objectList.M_GetIterator(iter);
WHILE iter.pNode > 0 AND_THEN iter.pNode^.P_pObject > 0 DO
	pObject := iter.pNode^.P_pObject;
	id := pObject^.P_nObjectID;
	a_pObjects[id] := 0;
	pObject^.M_ClearAllProps(TRUE);
	CASE pObject^.P_eObjectType OF
		E_ObjectType.OBJECTTYPE_Cartridge:
			pCartridge := pObject;
			__DELETE(pCartridge);
		E_ObjectType.OBJECTTYPE_FlipTube:
			pFlipTube := pObject;
			__DELETE(pFlipTube);
		E_ObjectType.OBJECTTYPE_Mtp:
			pMtp := pObject;
			__DELETE(pMtp);
		E_ObjectType.OBJECTTYPE_Needle:
			pNeedle := pObject;
			__DELETE(pNeedle);
		E_ObjectType.OBJECTTYPE_Nozzle:
			pNozzle := pObject;
			__DELETE(pNozzle);		
		E_ObjectType.OBJECTTYPE_pHElectrodeCap:
			pPHElectrodeCap := pObject;
			__DELETE(pPHElectrodeCap);
		E_ObjectType.OBJECTTYPE_Point:
			pPoint := pObject;
			__DELETE(pPoint);
		E_ObjectType.OBJECTTYPE_Port:
			pPort := pObject;
			__DELETE(pPort);
		E_ObjectType.OBJECTTYPE_Septum:
			pSeptum := pObject;
			__DELETE(pSeptum);
		E_ObjectType.OBJECTTYPE_Slide:
			pSlide := pObject;
			__DELETE(pSlide);
		E_ObjectType.OBJECTTYPE_SpotArray:
			pSpotArray := pObject;
			__DELETE(pSpotArray);
		(*E_ObjectType.OBJECTTYPE_SpotPattern:
			pSpotPattern := pObject;
			__DELETE(pSpotPattern);*)
		E_ObjectType.OBJECTTYPE_Stamp:
			pStamp := pObject;
			__DELETE(pStamp);
		E_ObjectType.OBJECTTYPE_Tip:
			pTip := pObject;
			__DELETE(pTip);
		E_ObjectType.OBJECTTYPE_TargetTray:
			pTray := pObject;
			__DELETE(pTray);
		E_ObjectType.OBJECTTYPE_Vial:
			pVial := pObject;
			__DELETE(pVial);
		E_ObjectType.OBJECTTYPE_VialClosed:
			pVialClosed := pObject;
			__DELETE(pVialClosed);
		(*E_ObjectType.OBJECTTYPE_Wafer:
			pWafer := pObject;
			__DELETE(pWafer);	*)
	END_CASE
	iter.M_Increment();
END_WHILE

objectList.M_Clear();
fbIdPool.M_Reset();
deviceList.M_Clear();

fbConfiguration.M_Deactivate();

FOR i := 1 TO cMaxMzHeads BY 1 DO
	aFbMultiZRef[i].M_DelConfig();
END_FOR
END_METHOD

METHOD M_DeleteObject : E_ErrorIdObjMgmt
VAR_INPUT
	nObjectID		: UINT;
END_VAR
VAR
	pDeviceNode	: POINTER TO FB_ObjCollectionNode;
	iter : FB_ObjCollectIterator;
END_VAR
//Existiert das Objekt ?
IF nObjectID > 0 AND nObjectID <= cMaxObjects THEN
	IF a_pObjects[nObjectId] > 0 THEN
		//Es können nur Objekte ohne Childs gelöscht werden
		IF NOT a_pObjects[nObjectId]^.P_bHasChilds THEN
			IF a_pObjects[nObjectId]^.M_bIsGroup(E_ObjectGroup.OBJECTGROUP_Device) THEN
				deviceList.M_GetIterator(iter);
				WHILE iter.pNode > 0 DO
					IF iter.pNode^.P_pObject = a_pObjects[nObjectId] THEN
						deviceList.M_ClearNode(iter.pNode);
						EXIT;
					END_IF
					iter.M_Increment();
				END_WHILE
			END_IF
		
			IF a_pObjects[nObjectId]^.P_nNotifyId > 0 THEN
				nCntNotifiIds := nCntNotifiIds - 1;
			END_IF
		
			IF a_pObjects[nObjectId]^.P_pParentObject > 0 THEN
				a_pObjects[nObjectId]^.P_pParentObject^.M_RemoveChild(a_pObjects[nObjectId]);
			ELSE
				IF a_pObjects[nObjectId]^.P_pObjCollectNode > 0 THEN
					a_pObjects[nObjectId]^.P_pObjCollectNode^.P_pOwnerColl^.M_ClearNode(a_pObjects[nObjectId]^.P_pObjCollectNode);
				END_IF
			END_IF
			
			IF a_pObjects[nObjectId]^.M_bIsGroup(E_ObjectGroup.OBJECTGROUP_MzTool) THEN
				fbConfiguration.M_Deactivate();
			END_IF
 			
			a_pObjects[nObjectId]^.M_ClearAllProps(FALSE);
		
			nCntObject := nCntObject - 1;
			
			CASE a_pObjects[nObjectId]^.P_eObjectType OF
				E_ObjectType.OBJECTTYPE_MZHead:
					nCntMZHead := nCntMZHead - 1;
				E_ObjectType.OBJECTTYPE_PiezoPip:
					nCntPiezoPip := nCntPiezoPip - 1;
				E_ObjectType.OBJECTTYPE_PassivPip:
					nCntPassivPip := nCntPassivPip - 1;
				E_ObjectType.OBJECTTYPE_pHElectrode:
					nCntpHElectrode := nCntpHElectrode - 1;
				E_ObjectType.OBJECTTYPE_pHElectrodeCap:
					pPHElectrodeCap := a_pObjects[nObjectId];
					__DELETE(pPHElectrodeCap);
				E_ObjectType.OBJECTTYPE_pHElectrodeCapRack:
					nCntpHElectrodeCapRack := nCntpHElectrodeCapRack - 1;
				E_ObjectType.OBJECTTYPE_PowderPip:
					nCntPowderPip := nCntPowderPip - 1;
				E_ObjectType.OBJECTTYPE_MultiCartHolder:
					nCntMultiCartHolder := nCntMultiCartHolder - 1;
				E_ObjectType.OBJECTTYPE_HybridDispenser:
					nCntHybridDispenser := nCntHybridDispenser - 1;
				E_ObjectType.OBJECTTYPE_CartDispenser:
					nCntCartDispenser := nCntCartDispenser - 1;
				E_ObjectType.OBJECTTYPE_CartDispStirrer:
					nCntCartDispStirrer := nCntCartDispStirrer - 1;
				E_ObjectType.OBJECTTYPE_CartHolder:
					nCntCartHolder := nCntCartHolder - 1;
				E_ObjectType.OBJECTTYPE_Camera:
					nCntCamera := nCntCamera - 1;
				E_ObjectType.OBJECTTYPE_ZSensor:
					nCntZLevelSensor := nCntZLevelSensor - 1;
				E_ObjectType.OBJECTTYPE_StampSupport:
					nCntStampSupport := nCntStampSupport - 1;
				E_ObjectType.OBJECTTYPE_Luer:
					nCntLuer := nCntLuer - 1;
				E_ObjectType.OBJECTTYPE_TrayTransporter:
					nCntTrayTransporter := nCntTrayTransporter - 1;
				E_ObjectType.OBJECTTYPE_TriplePip:
					nCntTriplePip := nCntTriplePip - 1;
				E_ObjectType.OBJECTTYPE_VacuumHandler:
					nCntVacuumHandler := nCntVacuumHandler - 1;
				E_ObjectType.OBJECTTYPE_Workplate:
					nCntWorkplate := nCntWorkplate - 1;
				E_ObjectType.OBJECTTYPE_TipCleaner:
					nCntTipCleaner := nCntTipCleaner - 1;
				E_ObjectType.OBJECTTYPE_TipCleanerGen2:
					nCntTipCleanerGen2 := nCntTipCleanerGen2 - 1;
				E_ObjectType.OBJECTTYPE_TipCalibrator:
					nCntTipCalibrator := nCntTipCalibrator - 1;
				E_ObjectType.OBJECTTYPE_TitrationTool:
					nCntTitrationTool := nCntTitrationTool - 1;
				E_ObjectType.OBJECTTYPE_WashStation:
					nCntWashStation := nCntWashStation - 1;
				E_ObjectType.OBJECTTYPE_LiquidReserve:
					nCntLiquidReserve := nCntLiquidReserve - 1;
				E_ObjectType.OBJECTTYPE_DryPad:
					nCntDrayPad := nCntDrayPad - 1;
				E_ObjectType.OBJECTTYPE_Stroboscope:
					nCntStroboscope := nCntStroboscope - 1;
				E_ObjectType.OBJECTTYPE_MtpHolder:
					nCntMtpHolder := nCntMtpHolder - 1;
				E_ObjectType.OBJECTTYPE_SubstHolder:
					nCntSubstHolder := nCntSubstHolder - 1;
				E_ObjectType.OBJECTTYPE_SubstHolderUnistat:
					nCntSubstHolderUnistat := nCntSubstHolderUnistat - 1;
				E_ObjectType.OBJECTTYPE_StampMagazine:
					nCntStampMagazine := nCntStampMagazine - 1;
				E_ObjectType.OBJECTTYPE_InkStation:
					nCntInkStation := nCntInkStation - 1;
				E_ObjectType.OBJECTTYPE_PowderStation:
					nCntPowderStation := nCntPowderStation - 1;
				E_ObjectType.OBJECTTYPE_Reactor:
					nCntReactor := nCntReactor - 1;
				E_ObjectType.OBJECTTYPE_TargetTray:
					pTray := a_pObjects[nObjectId];
					__DELETE(pTray);
				E_ObjectType.OBJECTTYPE_SpotArray:
					pSpotArray := a_pObjects[nObjectId];
					__DELETE(pSpotArray);
				E_ObjectType.OBJECTTYPE_Mtp:
					pMtp := a_pObjects[nObjectId];
					__DELETE(pMtp);
				E_ObjectType.OBJECTTYPE_Slide:
					pSlide := a_pObjects[nObjectId];
					__DELETE(pSlide);
				(*E_ObjectType.OBJECTTYPE_Wafer:
					pWafer := a_pObjects[nObjectId];
					__DELETE(pWafer);	*)				
				E_ObjectType.OBJECTTYPE_Point:
					pPoint := a_pObjects[nObjectId];
					__DELETE(pPoint);
				E_ObjectType.OBJECTTYPE_Diluter:
					fbConfiguration.M_Deactivate();
					nCntDiluter := nCntDiluter - 1;
				E_ObjectType.OBJECTTYPE_Diluter3Inputs:
					fbConfiguration.M_Deactivate();
					nCntDiluter3Inputs := nCntDiluter3Inputs - 1;
				(*E_ObjectType.OBJECTTYPE_SpotPattern:
					pSpotPattern := a_pObjects[nObjectId];
					__DELETE(pSpotPattern);*)
				E_ObjectType.OBJECTTYPE_DeloDot:
					nCntDeloDot := nCntDeloDot - 1;
				E_ObjectType.OBJECTTYPE_Exposure:
					nCntExposure := nCntExposure - 1;
				E_ObjectType.OBJECTTYPE_Stamp:
					pStamp := a_pObjects[nObjectId];
					__DELETE(pStamp);
				E_ObjectType.OBJECTTYPE_Needle:
					pNeedle := a_pObjects[nObjectId];
					__DELETE(pNeedle);
				E_ObjectType.OBJECTTYPE_Tip:
					pTip := a_pObjects[nObjectId];
					__DELETE(pTip);
				E_ObjectType.OBJECTTYPE_Vial:
					pVial := a_pObjects[nObjectId];
					__DELETE(pVial);
				E_ObjectType.OBJECTTYPE_VialClosed:
					pVialClosed := a_pObjects[nObjectId];
					__DELETE(pVialClosed);
				E_ObjectType.OBJECTTYPE_Septum:
					pSeptum := a_pObjects[nObjectId];
					__DELETE(pSeptum);
				E_ObjectType.OBJECTTYPE_Cartridge:
					pCartridge := a_pObjects[nObjectId];
					__DELETE(pCartridge);
				E_ObjectType.OBJECTTYPE_Port:
					pPort := a_pObjects[nObjectId];
					__DELETE(pPort);
				E_ObjectType.OBJECTTYPE_FlipTube:
					pFlipTube := a_pObjects[nObjectId];
					__DELETE(pFlipTube);
				E_ObjectType.OBJECTTYPE_SeptumWaste:
					nCntSeptumWaste := nCntSeptumWaste - 1;
				E_ObjectType.OBJECTTYPE_NeedleRack:
					nCntNeedleRack := nCntNeedleRack - 1;
				E_ObjectType.OBJECTTYPE_TipRack:
					nCntTipRack := nCntTipRack - 1;
				E_ObjectType.OBJECTTYPE_FlipTubeRack:
					nCntFlipTubeRack := nCntFlipTubeRack - 1;
				E_ObjectType.OBJECTTYPE_SeptumRack:
					nCntSeptumRack := nCntSeptumRack - 1;
				E_ObjectType.OBJECTTYPE_VialRack:
					nCntVialRack := nCntVialRack - 1;
				E_ObjectType.OBJECTTYPE_PortRack:
					nCntPortRack := nCntPortRack - 1;
				E_ObjectType.OBJECTTYPE_Nozzle:
					fbConfiguration.M_Deactivate();
					pNozzle := a_pObjects[nObjectId];
					__DELETE(pNozzle);
				E_ObjectType.OBJECTTYPE_SinglePiezoHolder:
					nCntSinglePiezoHolder := nCntSinglePiezoHolder - 1;
				E_ObjectType.OBJECTTYPE_TwinPiezoHolder:
					nCntTwinPiezoHolder := nCntTwinPiezoHolder - 1;
				E_ObjectType.OBJECTTYPE_HighVoltTray:
					nCntHighVoltTray := nCntHighVoltTray - 1;
				E_ObjectType.OBJECTTYPE_SolenoidPip:
					nCntSolenoidPip := nCntSolenoidPip - 1;
				E_ObjectType.OBJECTTYPE_Extruder:
					nCntExtruder := nCntExtruder - 1;
				E_ObjectType.OBJECTTYPE_TwinExtruder:
					nCntTwinExtruder := nCntTwinExtruder - 1;
				E_ObjectType.OBJECTTYPE_VermesDisp:
					nCntVermesDisp := nCntVermesDisp - 1;
				E_ObjectType.OBJECTTYPE_WorkplateCamera:
					nCntWorkplateCamera := nCntWorkplateCamera - 1;
				E_ObjectType.OBJECTTYPE_DummyTool:
					nCntDummyTool := nCntDummyTool - 1;
				E_ObjectType.OBJECTTYPE_CustomUnitType1:
					nCntCustomUnitType1 := nCntCustomUnitType1 - 1;
				E_ObjectType.OBJECTTYPE_CustomUnitType2:
					nCntCustomUnitType2 := nCntCustomUnitType2 - 1;
				E_ObjectType.OBJECTTYPE_Gripper:
					nCntGripper := nCntGripper - 1;
				E_ObjectType.OBJECTTYPE_PickPlacePip:
					nCntPickPlacePip := nCntPickPlacePip - 1;
				E_ObjectType.OBJECTTYPE_Stacker:
					nCntStacker := nCntStacker - 1;
			END_CASE
			a_pObjects[nObjectId] := 0;
			//ObjectID wieder freigeben
			fbIdPool.M_ReleaseId(nObjectId);
		ELSE
			M_DeleteObject := E_ErrorIdObjMgmt.ERRORID_ObjectHasChilds;
		END_IF
	ELSE
		M_DeleteObject := E_ErrorIdObjMgmt.ERRORID_InvalidObjectId;
	END_IF
END_IF
END_METHOD

METHOD M_GetChangedObjId : UINT
VAR_INPUT
END_VAR
IF hList.nCount > 0 THEN
	fbList.A_GetTail(hList:= hList);
	{IF hasvalue (RegisterSize, '32')}
	M_GetChangedObjId := UDINT_TO_UINT(fbList.getValue);
	{ELSE}
	M_GetChangedObjId := ULINT_TO_UINT(fbList.getValue);
	{END_IF}
	fbList.A_RemoveTailValue(hList:= hList);
END_IF
END_METHOD

METHOD M_GetCoHead : POINTER TO FB_MzHead
VAR_INPUT
	pMzHead : POINTER TO FB_MzHead;
END_VAR

VAR
	i : UINT;
END_VAR
FOR i:= 1 TO nCntMZHead BY 1 DO
	IF ADR(afbMzHead[i]) <> pMzHead THEN
		IF afbMzHead[i].P_eObjectType = E_ObjectType.OBJECTTYPE_MZHead THEN
			IF afbMzHead[i].P_pXDrive = pMzHead^.P_pXDrive THEN
				M_GetCoHead := ADR(afbMzHead[i]);
			END_IF
		END_IF
	END_IF
END_FOR
END_METHOD

METHOD M_GetConfigCheckSum : UINT
VAR_INPUT
END_VAR

VAR
	nObjectCounter 	: UINT;
	wPrevious 		: WORD := 16#FFFF;
	iter			: FB_ObjCollectIteratorDeep;
	nLevel			: UINT;
	nObjType		: UINT;
	nNoOfProps		: UINT;
	nParentSlotNr	: UINT;
END_VAR
objectList.M_GetIterator(iter);
WHILE iter.pNode > 0 AND_THEN iter.pNode^.P_pObject > 0 DO
	
	nParentSlotNr := iter.pNode^.P_pObject^.P_nParentSlotNr;
	wPrevious := F_DATA_TO_CRC16_CCITT(ADR(nParentSlotNr),SIZEOF(nParentSlotNr),wPrevious);

	nLevel := iter.pNode^.M_GetLevel(0);
	wPrevious := F_DATA_TO_CRC16_CCITT(ADR(nLevel),SIZEOF(nLevel),wPrevious); 

	nObjType := iter.pNode^.P_pObject^.P_eObjectType;
	wPrevious := F_DATA_TO_CRC16_CCITT(ADR(nObjType),SIZEOF(nObjType),wPrevious);

	nNoOfProps := iter.pNode^.P_pObject^.P_nNoOfProps;
	wPrevious := F_DATA_TO_CRC16_CCITT(ADR(nNoOfProps),SIZEOF(nNoOfProps),wPrevious);

	iter.M_Increment();
END_WHILE
M_GetConfigCheckSum := WORD_TO_UINT(wPrevious);
END_METHOD

METHOD M_GetDevice : I_Device
VAR_INPUT
	nObjectId : UINT;
END_VAR

VAR
	pActiveTarget : POINTER TO FB_ActiveTarget;
	pMzToolBase	: POINTER TO FB_MzBase;
	pDiluter : POINTER TO FB_Diluter; 
END_VAR
IF M_ObjIsDevice(nObjectId) THEN
	M_GetDevice := a_pObjects[nObjectId]^.M_GetDevice();
END_IF
END_METHOD

METHOD M_GetObjIdFromGCodeTargetNr : UINT
VAR_INPUT
	nTargetNr : UINT;
END_VAR
END_METHOD

METHOD M_GetObjIdStream : ERRORID
VAR_INPUT
	aData : REFERENCE TO ARRAY[0..999] OF UINT;
END_VAR

VAR
	iter : FB_ObjCollectIteratorDeep;
	i : UINT;
END_VAR
objectList.M_GetIterator(iter);
WHILE iter.pNode > 0 AND_THEN iter.pNode^.P_pObject > 0 DO
	IF i > 999 THEN
		M_GetObjIdStream := 333;
		RETURN;	
	END_IF
	aData[i] := iter.pNode^.P_pObject^.P_nObjectID;
	i := i + 1;
	iter.M_Increment();
END_WHILE
END_METHOD

METHOD M_GetObjPointer : POINTER TO FB_Object
VAR_INPUT
	nObjectId : UINT;
END_VAR
IF nObjectId > 0 AND nObjectId <= cMaxObjects THEN
	IF a_pObjects[nObjectId]^.P_nObjectID = nObjectId THEN
		M_GetObjPointer := a_pObjects[nObjectId];
	END_IF
END_IF
END_METHOD

METHOD M_GetObjType : E_ObjectType
VAR_INPUT
	ObjectId	: UINT;
END_VAR
IF ObjectId > 0 AND ObjectId <= cMaxObjects AND_THEN a_pObjects[ObjectId] > 0 THEN
	M_GetObjType := a_pObjects[ObjectId]^.P_eObjectType;
ELSE
	M_GetObjType := E_ObjectType.OBJECTTYPE_UNDEFINED;
END_IF
END_METHOD

METHOD M_GetTipCleaner : POINTER TO FB_TargetBase
VAR_INPUT
END_VAR
//Es wird davon ausgegangen, dass es nur einen TipCleaner in einer Konfiguration gibt.
IF afbTipCleaner[1].P_nObjectID > 0 THEN
	M_GetTipCleaner := ADR(afbTipCleaner[1]);
ELSIF afbTipCleanerGen2[1].P_nObjectID > 0 THEN
	M_GetTipCleaner := ADR(afbTipCleanerGen2[1]);
END_IF
END_METHOD

METHOD M_GetTopHead : POINTER TO FB_MzHead

VAR
	i : UINT;
END_VAR
FOR i:= 1 TO nCntMZHead BY 1 DO
	IF afbMzHead[i].P_bIsTopHead THEN
		M_GetTopHead := ADR(afbMzHead[i]);
		RETURN;
	END_IF
END_FOR
END_METHOD

METHOD M_Init : BOOL
VAR_INPUT
END_VAR

VAR
	i	: UINT;	//allg. Zählveriable
END_VAR
fbIdPool.M_Reset();

F_CreateLinkedListHnd( ADR( nodes ), SIZEOF( nodes ), hList );

bIsInitialized := TRUE;
END_METHOD

METHOD M_MoveObject : ERRORID
VAR_INPUT
	pObject : POINTER TO FB_Object;
	pDestObject : POINTER TO FB_Object;
	nDestSlotNr	: UINT;
END_VAR

VAR
	pSlot : POINTER TO FB_Slot;
END_VAR
//Verschiebt ein Objekt zu einem neuen Objekt oder zu einem anderen Slot.
IF pObject > 0 THEN
	IF pObject^.P_pParentObject > 0 AND_THEN pDestObject > 0 THEN
		IF nDestSlotNr > 0 THEN
			pSlot := pDestObject^.M_GetSlot(nDestSlotNr);
			IF pSlot > 0 THEN
				IF pSlot^.P_pChild > 0 THEN
					M_MoveObject := E_ErrorIdObjMgmt.ERRORID_DestinationSlotNotFree;
					RETURN;
				END_IF
			ELSE
				M_MoveObject := E_ErrorIdObjMgmt.ERRORID_InvalidDestinationSlot;
				RETURN;
			END_IF
		END_IF
		M_MoveObject := pObject^.P_pParentObject^.M_RemoveChild(pObject);
		IF M_MoveObject = 0 THEN
			M_MoveObject := pDestObject^.M_AddChild(pObject,nDestSlotNr,-1);
			//M_SetObjChange(pObject^.P_nObjectID);
			stObjectHasMoved.ObjectId := pObject^.P_nObjectID;
			stObjectHasMoved.DestObjId := pDestObject^.P_nObjectID;
			stObjectHasMoved.DestSlotNr := nDestSlotNr;
			stObjectHasMoved.ChangeCounter := stObjectHasMoved.ChangeCounter + 1;
		END_IF
	ELSE
		M_MoveObject := E_ErrorIdObjMgmt.ERRORID_InvalidObject;
	END_IF
ELSE
	M_MoveObject := E_ErrorIdObjMgmt.ERRORID_InvalidObject;
END_IF
END_METHOD

METHOD M_ObjIsArray : BOOL
VAR_INPUT
	nObjectId	: UINT;
END_VAR
IF nObjectId > 0 AND nObjectId <= cMaxObjects THEN
	IF (a_pObjects[nObjectId]^.P_eObjectGroup AND E_ObjectGroup.OBJECTGROUP_Array) = E_ObjectGroup.OBJECTGROUP_Array THEN
		M_ObjIsArray := TRUE;
	END_IF
END_IF
END_METHOD

METHOD M_ObjIsDevice : BOOL
VAR_INPUT
	nObjectId	: UINT;
END_VAR
IF nObjectId > 0 AND nObjectId <= cMaxObjects THEN
	IF a_pObjects[nObjectId]^.M_bIsGroup(E_ObjectGroup.OBJECTGROUP_Device) THEN
		M_ObjIsDevice := TRUE;
	END_IF
END_IF
END_METHOD

METHOD M_ObjIsGCodeTool : BOOL
VAR_INPUT
	nObjectId	: UINT;
END_VAR
IF nObjectId > 0 AND nObjectId <= cMaxObjects THEN
	IF (a_pObjects[nObjectId]^.P_eObjectGroup AND E_ObjectGroup.OBJECTGROUP_GCodeTool) = E_ObjectGroup.OBJECTGROUP_GCodeTool THEN
		M_ObjIsGCodeTool := TRUE;
	END_IF
END_IF
END_METHOD

METHOD M_ObjIsMzTool : BOOL
VAR_INPUT
	nObjectId	: UINT;
END_VAR
IF nObjectId > 0 AND nObjectId <= cMaxObjects THEN
	IF (a_pObjects[nObjectId]^.P_eObjectGroup AND E_ObjectGroup.OBJECTGROUP_MzTool) = E_ObjectGroup.OBJECTGROUP_MzTool THEN
		M_ObjIsMzTool := TRUE;
	END_IF
END_IF
END_METHOD

METHOD M_ObjIsPiece : BOOL
VAR_INPUT
	nObjectId	: UINT;
END_VAR
IF nObjectId > 0 AND nObjectId <= cMaxObjects THEN
	IF (a_pObjects[nObjectId]^.P_eObjectGroup AND E_ObjectGroup.OBJECTGROUP_Piece) = E_ObjectGroup.OBJECTGROUP_Piece THEN
		M_ObjIsPiece := TRUE;
	END_IF
END_IF
END_METHOD

METHOD M_ObjIsRack : BOOL
VAR_INPUT
	nObjectId	: UINT;
END_VAR
IF nObjectId > 0 AND nObjectId <= cMaxObjects THEN
	IF (a_pObjects[nObjectId]^.P_eObjectGroup AND E_ObjectGroup.OBJECTGROUP_Rack) = E_ObjectGroup.OBJECTGROUP_Rack THEN
		M_ObjIsRack := TRUE;
	END_IF
END_IF
END_METHOD

METHOD M_ObjIsTarget : BOOL
VAR_INPUT
	nObjectId	: UINT;
END_VAR
IF nObjectId > 0 AND nObjectId <= cMaxObjects THEN
	IF (a_pObjects[nObjectId]^.P_eObjectGroup AND E_ObjectGroup.OBJECTGROUP_Target) = E_ObjectGroup.OBJECTGROUP_Target THEN
		M_ObjIsTarget := TRUE;
	END_IF
END_IF
END_METHOD

METHOD M_RemoveObjChange
VAR_INPUT
	nObjectId : UINT;
END_VAR

VAR
	getPosPtr : POINTER TO T_LinkedListEntry;
END_VAR
fbList.A_FindNext(hList:= hList, putPosPtr:= 0, putValue:= UINT_TO_UDINT(nObjectId), getPosPtr=> getPosPtr);
IF fbList.bOk THEN //Eintrag vorhanden
	fbList.A_RemoveValueAtPosPtr(hList:= hList, putPosPtr := getPosPtr);
END_IF
END_METHOD

METHOD M_ResetCustomUnitType2
VAR_INPUT
END_VAR

VAR
	i : UINT;
END_VAR
FOR i := 1 TO nCntCustomUnitType2 DO
	 IF afbCustomUnitType2[i].P_bError THEN
		 afbCustomUnitType2[i].M_Reset();
	 END_IF
END_FOR
END_METHOD

METHOD M_SetObjChange
VAR_INPUT
	nObjectId : UINT;
END_VAR

VAR
	putValue : UDINT;
END_VAR
putValue := UINT_TO_UDINT(nObjectId);
//Checken, ob schon eingetragen
fbList.A_FindNext(hList:= hList, putPosPtr:= 0, putValue:= putValue);
IF NOT fbList.bOk THEN //Eintrag noch nicht vorhanden
	fbList.A_AddHeadValue(hList:= hList, putValue:= putValue);	
	nObjPropChangeCnt := nObjPropChangeCnt + 1;
END_IF
END_METHOD

METHOD M_SetParent : ERRORID
VAR_INPUT
END_VAR
END_METHOD

PROPERTY P_pDeviceCollection : POINTER TO FB_ObjCollection
GET
P_pDeviceCollection := ADR(deviceList);
END_GET
END_PROPERTY

PROPERTY P_pObjectCollection : POINTER TO FB_ObjCollection
GET
P_pObjectCollection := ADR(objectList);
END_GET
END_PROPERTY

END_FUNCTION_BLOCK

// ---- Configuration/FB_IdPool.TcPOU
FUNCTION_BLOCK FB_IdPool
VAR_INPUT
END_VAR
VAR_OUTPUT
END_VAR
VAR
	aNodes : ARRAY[1..cMaxObjects] OF ST_IdNode;
	pHead : POINTER TO ST_IdNode;
	pTail : POINTER TO ST_IdNode;
END_VAR

METHOD M_GetId : UINT
VAR_INPUT
END_VAR

VAR
	pNode : POINTER TO ST_IdNode;
END_VAR
IF pHead > 0 THEN
	pNode := pHead;
	M_GetId := pNode^.nId;
	IF pHead = pTail THEN //die letzte freie Id
		pHead := 0;
		pTail := 0;
	ELSE
		pHead := pNode^.pNext;
	END_IF
	memset(pNode,0,SIZEOF(ST_IdNode));
END_IF
END_METHOD

METHOD M_ReleaseId : BOOL
VAR_INPUT
	nId : UINT;
END_VAR
//Id in Benutzung?
IF nId >= 0 AND nId <= cMaxObjects AND_THEN aNodes[nId].nId = 0 THEN
	aNodes[nId].nId := nId;
	aNodes[nId].pNext := pHead;
	pHead := ADR(aNodes[nId]);
	M_ReleaseId := TRUE;
END_IF
END_METHOD

METHOD M_Reset : BOOL
VAR_INPUT
END_VAR

VAR
	i : UINT;
END_VAR
pHead := ADR(aNodes[1]);
pTail := ADR(aNodes[cMaxObjects]);
FOR i := 1 TO cMaxObjects BY 1 DO
	aNodes[i].nId := i;
	IF i < cMaxObjects THEN
		aNodes[i].pNext := ADR(aNodes[i+1]);
	ELSE
		aNodes[i].pNext := 0;
	END_IF
END_FOR
END_METHOD

END_FUNCTION_BLOCK

// ---- Objects/Pieces/FB_Cartridge.TcPOU
{attribute 'enable_dynamic_creation'}
FUNCTION_BLOCK FB_Cartridge EXTENDS FB_PieceBase
VAR_INPUT
END_VAR
VAR_OUTPUT
END_VAR
VAR
END_VAR

METHOD FB_init : BOOL
VAR_INPUT
	bInitRetains : BOOL; // if TRUE, the retain variables are initialized (warm start / cold start)
	bInCopyCode : BOOL;  // if TRUE, the instance afterwards gets moved into the copy code (online change)
END_VAR
eObjectType := E_ObjectType.OBJECTTYPE_Cartridge;
eObjectGroup := E_ObjectGroup.OBJECTGROUP_Piece;
END_METHOD

END_FUNCTION_BLOCK

// ---- Objects/Pieces/FB_FlipTube.TcPOU
{attribute 'enable_dynamic_creation'}
FUNCTION_BLOCK FB_FlipTube EXTENDS FB_PieceBase
VAR_INPUT
END_VAR
VAR_OUTPUT
END_VAR
VAR
	bIsOpen : BOOL;
	nTopLevel : DINT;
	nBottomLevel : DINT;	
END_VAR

METHOD FB_init : BOOL
VAR_INPUT
	bInitRetains : BOOL; // if TRUE, the retain variables are initialized (warm start / cold start)
	bInCopyCode : BOOL;  // if TRUE, the instance afterwards gets moved into the copy code (online change)
END_VAR
eObjectType := E_ObjectType.OBJECTTYPE_FlipTube;
eObjectGroup := E_ObjectGroup.OBJECTGROUP_Piece;
END_METHOD

METHOD M_GetAllProps : ERRORID
VAR_INPUT
	refCmdData : REFERENCE TO  ST_CmdData;
END_VAR
SUPER^.M_GetAllProps(refCmdData);
nCurrentPropIndex := nCurrentPropIndex + 1;
refCmdData.n32Data[nCurrentPropIndex] := BOOL_TO_DINT(bIsOpen);
nCurrentPropIndex := nCurrentPropIndex + 1;
refCmdData.n32Data[nCurrentPropIndex] := nTopLevel;
nCurrentPropIndex := nCurrentPropIndex + 1;
refCmdData.n32Data[nCurrentPropIndex] := nBottomLevel;
END_METHOD

{attribute 'object_name' := 'M_SetAllProps'}
METHOD M_SetAllProps : ERRORID
VAR_INPUT
	refCmdData	: REFERENCE TO ST_CmdData;
END_VAR
M_SetAllProps := SUPER^.M_SetAllProps(refCmdData);

IF M_SetAllProps > 0 THEN
	RETURN;
END_IF
nCurrentPropIndex := nCurrentPropIndex + 1;
nSpecPropIndex := nCurrentPropIndex;

bIsOpen := DINT_TO_BOOL(refCmdData.n32Data[nCurrentPropIndex]);
nCurrentPropIndex := nCurrentPropIndex + 1;
nTopLevel := refCmdData.n32Data[nCurrentPropIndex];
nCurrentPropIndex := nCurrentPropIndex + 1;
nBottomLevel := refCmdData.n32Data[nCurrentPropIndex];

nNoOfProps := nCurrentPropIndex + 1;
END_METHOD

METHOD M_SetSingleProp : ERRORID
VAR_INPUT
	refCmdData : REFERENCE TO  ST_CmdData;
END_VAR
IF refCmdData.aHeader[1] = nSpecPropIndex THEN
	bIsOpen := DINT_TO_BOOL(refCmdData.n32Data[0]);
ELSIF refCmdData.aHeader[1] + 1 = nSpecPropIndex THEN
	nTopLevel := refCmdData.n32Data[0];
ELSIF refCmdData.aHeader[1] + 2 = nSpecPropIndex THEN
	nBottomLevel := refCmdData.n32Data[0];
ELSE
	M_SetSingleProp := SUPER^.M_SetSingleProp(refCmdData);
END_IF
END_METHOD

PROPERTY P_bIsOpen : BOOL
GET
P_bIsOpen := bIsOpen;
END_GET
SET
bIsOpen := P_bIsOpen;
END_SET
END_PROPERTY

PROPERTY P_nBottomLevel : DINT
GET
P_nBottomLevel := nBottomLevel;
END_GET
END_PROPERTY

PROPERTY P_nTopLevel : DINT
GET
P_nTopLevel := nTopLevel;
END_GET
END_PROPERTY

END_FUNCTION_BLOCK

// ---- Objects/Pieces/FB_Needle.TcPOU
{attribute 'enable_dynamic_creation'}
FUNCTION_BLOCK FB_Needle EXTENDS FB_UsingPiece
VAR_INPUT
END_VAR
VAR_OUTPUT
END_VAR
VAR
	pSeptum : POINTER TO FB_PieceBase;
END_VAR

METHOD FB_init : BOOL
VAR_INPUT
	bInitRetains : BOOL; // if TRUE, the retain variables are initialized (warm start / cold start)
	bInCopyCode : BOOL;  // if TRUE, the instance afterwards gets moved into the copy code (online change)
END_VAR
bUsingPiece := TRUE;
eObjectType := E_ObjectType.OBJECTTYPE_Needle;
eObjectGroup := E_ObjectGroup.OBJECTGROUP_Piece;
END_METHOD

{attribute 'object_name' := 'M_ClearAllProps'}
METHOD M_ClearAllProps

VAR_INPUT
	bIgnoreParent : BOOL; //Es wird das gesamte OD gelöscht. -> Zeiger auf Parent nicht mehr gültig!
END_VAR
pSeptum := 0;
SUPER^.M_ClearAllProps(bIgnoreParent);
END_METHOD

PROPERTY P_pLatestChild : POINTER TO FB_PieceBase
GET
IF pSeptum > 0 THEN
	P_pLatestChild := pSeptum;	
ELSE
	P_pLatestChild := THIS;
END_IF
END_GET
END_PROPERTY

PROPERTY P_pSeptum : POINTER TO FB_PieceBase
GET
P_pSeptum := pSeptum;
END_GET
SET
pSeptum := P_pSeptum;
END_SET
END_PROPERTY

END_FUNCTION_BLOCK

// ---- Objects/Pieces/FB_pHElectrodeCap.TcPOU
{attribute 'enable_dynamic_creation'}
FUNCTION_BLOCK FB_pHElectrodeCap EXTENDS FB_PieceBase
VAR_INPUT
END_VAR
VAR_OUTPUT
END_VAR
VAR
END_VAR

METHOD FB_init : BOOL
VAR_INPUT
	bInitRetains : BOOL; // if TRUE, the retain variables are initialized (warm start / cold start)
	bInCopyCode : BOOL;  // if TRUE, the instance afterwards gets moved into the copy code (online change)
END_VAR
eObjectType := E_ObjectType.OBJECTTYPE_pHElectrodeCap;
eObjectGroup := E_ObjectGroup.OBJECTGROUP_Piece;
END_METHOD

END_FUNCTION_BLOCK

// ---- Objects/Targets/Passive/FB_Point.TcPOU
{attribute 'enable_dynamic_creation'}
FUNCTION_BLOCK FB_Point EXTENDS FB_TargetBase
VAR_INPUT
END_VAR
VAR_OUTPUT
END_VAR
VAR
END_VAR

METHOD FB_init : BOOL
VAR_INPUT
	bInitRetains : BOOL; // if TRUE, the retain variables are initialized (warm start / cold start)
	bInCopyCode : BOOL;  // if TRUE, the instance afterwards gets moved into the copy code (online change)
END_VAR
eObjectType := E_ObjectType.OBJECTTYPE_Point;
eObjectGroup := E_ObjectGroup.OBJECTGROUP_Target;
END_METHOD

METHOD M_AddChild : ERRORID
VAR_INPUT
	pObject : POINTER TO FB_Object;
	nSlotNr	: UINT;
	nIndex 	: INT;
END_VAR
//Kann folgende Objekte aufnehmen:
//Point
IF pObject <> 0 THEN
	IF pObject^.P_eObjectType = E_ObjectType.OBJECTTYPE_Point OR pObject^.P_eObjectType = E_ObjectType.OBJECTTYPE_SpotArray Then
		M_AddChild := SUPER^.M_AddChild(pObject,nSlotNr,nIndex);
	ELSE
		M_AddChild := E_ErrorIdObjMgmt.ERRORID_InvalidParentObject;
	END_IF
ELSE
	M_AddChild := E_ErrorIdObjMgmt.ERRORID_InvalidParentObject;
END_IF
END_METHOD

END_FUNCTION_BLOCK

// ---- Objects/Pieces/FB_Port.TcPOU
{attribute 'enable_dynamic_creation'}
FUNCTION_BLOCK FB_Port EXTENDS FB_PieceBase
VAR_INPUT
END_VAR
VAR_OUTPUT
END_VAR
VAR
END_VAR

METHOD FB_init : BOOL
VAR_INPUT
	bInitRetains : BOOL; // if TRUE, the retain variables are initialized (warm start / cold start)
	bInCopyCode : BOOL;  // if TRUE, the instance afterwards gets moved into the copy code (online change)
END_VAR
eObjectType := E_ObjectType.OBJECTTYPE_Port;
eObjectGroup := E_ObjectGroup.OBJECTGROUP_Piece;
END_METHOD

END_FUNCTION_BLOCK

// ---- Objects/Pieces/FB_Septum.TcPOU
{attribute 'enable_dynamic_creation'}
FUNCTION_BLOCK FB_Septum EXTENDS FB_UsingPiece
VAR_INPUT
END_VAR
VAR_OUTPUT
END_VAR
VAR
	pVial : POINTER TO FB_Vial;
END_VAR

METHOD FB_init : BOOL
VAR_INPUT
	bInitRetains : BOOL; // if TRUE, the retain variables are initialized (warm start / cold start)
	bInCopyCode : BOOL;  // if TRUE, the instance afterwards gets moved into the copy code (online change)
END_VAR
bUsingPiece := TRUE;
eObjectType := E_ObjectType.OBJECTTYPE_Septum;
eObjectGroup := E_ObjectGroup.OBJECTGROUP_Piece;
END_METHOD

{attribute 'object_name' := 'M_ClearAllProps'}
METHOD M_ClearAllProps

VAR_INPUT
	bIgnoreParent : BOOL; //Es wird das gesamte OD gelöscht. -> Zeiger auf Parent nicht mehr gültig!
END_VAR
pVial := 0;
SUPER^.M_ClearAllProps(bIgnoreParent);
END_METHOD

PROPERTY P_pVial : POINTER TO FB_PieceBase
GET
P_pVial := pVial;
END_GET
SET
pVial := P_pVial;
END_SET
END_PROPERTY

END_FUNCTION_BLOCK

// ---- Objects/Targets/Passive/FB_Slide.TcPOU
{attribute 'enable_dynamic_creation'}
FUNCTION_BLOCK FB_Slide EXTENDS FB_TargetBase
VAR_INPUT
END_VAR
VAR_OUTPUT
END_VAR
VAR
	///Spec-Properties TODO: rauslöschen
	(*
	nNoOfSpecPoints: USINT;
	stMark1: ST_3DPoint;
	stMark2: ST_3DPoint;
	stMark1Act: ST_3DPoint;
	stMark2Act: ST_3DPoint;*)
	
	//neue Slide Variablen
	stMarker1Position	: ST_3DPoint;
	stCamOffsetMarker1	: ST_3DPoint;
	stCamOffsetMarker2	: ST_3DPoint;
	rTargetRot			: REAL;			//Winkel * 1000
	
	//ALT: 
	
	lrAngle				: LREAL;
	//bIsAligned			: BOOL;	
END_VAR

METHOD FB_init : BOOL
VAR_INPUT
	bInitRetains : BOOL; // if TRUE, the retain variables are initialized (warm start / cold start)
	bInCopyCode : BOOL;  // if TRUE, the instance afterwards gets moved into the copy code (online change)
END_VAR
eObjectType := E_ObjectType.OBJECTTYPE_Slide;
eObjectGroup := E_ObjectGroup.OBJECTGROUP_Target;
END_METHOD

METHOD M_AddChild : ERRORID
VAR_INPUT
	pObject : POINTER TO FB_Object;
	nSlotNr	: UINT;
	nIndex 	: INT;
END_VAR
//Kann folgende Objekte aufnehmen:
IF pObject > 0 THEN
	IF pObject^.P_eObjectType = E_ObjectType.OBJECTTYPE_Point OR
		pObject^.P_eObjectType = E_ObjectType.OBJECTTYPE_Slide OR
		pObject^.P_eObjectType = E_ObjectType.OBJECTTYPE_Mtp OR
		(*pObject^.P_eObjectType = E_ObjectType.OBJECTTYPE_SpotPattern OR*)
		pObject^.P_eObjectType = E_ObjectType.OBJECTTYPE_SpotArray
		(*pObject^.P_eObjectType = E_ObjectType.OBJECTTYPE_TargetGroup OR
		pObject^.P_eObjectType = E_ObjectType.OBJECTTYPE_Wafer*) THEN
		M_AddChild := SUPER^.M_AddChild(pObject,nSlotNr,nIndex);
	ELSE
		M_AddChild := E_ErrorIdObjMgmt.ERRORID_InvalidParentObject;
	END_IF
ELSE
	M_AddChild := E_ErrorIdObjMgmt.ERRORID_InvalidParentObject;
END_IF
END_METHOD

METHOD M_Align : ST_3DPoint
VAR_INPUT
	stPos: ST_3DPoint;
END_VAR
VAR_OUTPUT
	lrAngle: LREAL;
END_VAR
VAR
	stPosTmp: ST_3DPoint;
END_VAR
//lrAngle := THIS^.lrAngle;
END_METHOD

METHOD M_CalcAngle : ERRORID
VAR_INPUT
END_VAR
(*IF bIsAligned THEN
	//Falls ein Fehler bei der Berechnung auftritt, wird "bIsAligned" zurückgesetzt
	lrAngle := F_GetTwoLineAngle(stMark1,stMark2,stMark1Act, stMark2Act);
	IF lrAngle = 9999.9 THEN
		bIsAligned := FALSE;
		lrAngle := 0.0;
	END_IF
ELSE
	lrAngle := 0.0;
END_IF*)
END_METHOD

METHOD M_ClearAllProps
VAR_INPUT
	bIgnoreParent : BOOL; //Es wird das gesamte OD gelöscht. -> Zeiger auf Parent nicht mehr gültig!
END_VAR
SUPER^.M_ClearAllProps(bIgnoreParent);
//bIsAligned:= FALSE;
END_METHOD

METHOD M_GetAbsPos : ST_3DPoint
VAR_INPUT
	pChildPos	: POINTER TO ST_3DPoint;
	eTargetRef 	: E_TargetRef;
	nParam1		: UINT;
 	nParam2		: UINT;
	nParam3		: USINT;
	nZLevel		: USINT;
END_VAR
VAR_OUTPUT
	nErrorId 	: ERRORID;
	lrAngle		: LREAL;

END_VAR
VAR
	stLocPos: ST_3DPoint;
	stLocPosAligned: ST_3DPoint;
	stNull: ST_3DPoint;

	nState_SlideGetAbsPos	: USINT;
END_VAR
(*stLocPos.Z := stLocPos.Z + stDimension.Height + rZOffset;
CASE eTargetRef OF
	E_TargetRef.TARGETREF_LeftBottom:
		;
	E_TargetRef.TARGETREF_LeftTop:
		stLocPos.Y := stLocPos.Y + stDimension.Depth;
	E_TargetRef.TARGETREF_RightBottom:
		stLocPos.X := stLocPos.X + stDimension.Width;
	E_TargetRef.TARGETREF_RightTop:
		stLocPos.X := stLocPos.X + stDimension.Width;
		stLocPos.Y := stLocPos.Y + stDimension.Depth;
	E_TargetRef.TARGETREF_Center:
		stLocPos.X := stLocPos.X + stDimension.Width / 2.0;
		stLocPos.Y := stLocPos.Y + stDimension.Depth / 2.0;
	(*E_TargetRef.TARGETREF_SpecPoint:
		IF nNoOfSpecPoints = 2 THEN
			IF nParam1 = 1 THEN	//Mark1
				stLocPos := F_Add3DPoints(stLocPos,stMark1);
			ELSIF nParam1 = 2 THEN	//Mark2
				stLocPos := F_Add3DPoints(stLocPos,stMark2);
			ELSE
				nErrorId := E_ErrorIdCmd.ERRORID_InvalidTargetPointNr;
			END_IF	
		ELSE
			nErrorId := E_ErrorIdCmd.ERRORID_InvalidTargetPointNr;	
		END_IF*)
	
ELSE
	nErrorId := E_ErrorIdCmd.ERRORID_InvalidTargetPointRef;
END_CASE

IF nErrorId > 0 THEN
	RETURN;
END_IF

//Marker 1 Position wird noch nicht übermittelt von GUI. TODO: Wenn Übermittlung funktioniert, dann raus löschen
stMarker1Position.X := 4500;
stMarker1Position.Y := 4500;
stLocPosAligned := stLocPos;

IF rTargetRot <> 0  THEN	//Im Grunde müssten sich die Marken genauso drehen lassen
	//Offset
	lrAngle := rTargetRot/1000;
	stLocPosAligned.X := stLocPosAligned.X + stCamOffsetMarker1.X;
	stLocPosAligned.Y := stLocPosAligned.Y + stCamOffsetMarker1.Y;
	//Drehen
	stLocPosAligned := F_RotatePoint(stLocPosAligned,stNull,THIS^.lrAngle);
END_IF

stLocPos := F_Add3DPoints(stLocPos,stRelPos);
stLocPosAligned := F_Add3DPoints(stLocPosAligned,stRelPos);

IF pChildPos > 0 THEN
	IF rTargetRot <> 0 THEN
		pChildPos^ := F_RotatePoint(pChildPos^,stNull,THIS^.lrAngle);
	END_IF
	
	pChildPos^.X := pChildPos^.X + stLocPosAligned.X - stLocPos.X;
	pChildPos^.Y := pChildPos^.Y + stLocPosAligned.Y - stLocPos.Y;

	stLocPos.X := pChildPos^.X + stLocPos.X;
	stLocPos.Y := pChildPos^.Y + stLocPos.Y;
	stLocPos.Z := pChildPos^.Z + stLocPos.Z;
ELSE
	stLocPos := stLocPosAligned;
END_IF

IF pParentTarget > 0 THEN
	IF pParentSlot > 0 THEN
 		stLocPos := pParentTarget^.M_GetAbsPos(pChildPos := ADR(stLocPos), eTargetRef:= E_TargetRef.TARGETREF_Slot,
													nParam1:= pParentSlot^.P_nNr,
													nParam2:= 0, nParam3:= 0,nZLevel:= 0,
													lrAngle => lrAngle, nErrorId=> nErrorId);
	ELSE
 		stLocPos := pParentTarget^.M_GetAbsPos(pChildPos := ADR(stLocPos), eTargetRef:= E_TargetRef.TARGETREF_LeftBottom,
													nParam1:= 0,
													nParam2:= 0, nParam3:= 0,nZLevel:= 0,
													lrAngle => lrAngle, nErrorId=> nErrorId);
	END_IF
END_IF

IF nErrorId > 0 THEN
	RETURN;
END_IF

IF rTargetRot <> 0 THEN
	lrAngle := lrAngle + THIS^.lrAngle;	
END_IF

M_GetAbsPos := stLocPos;
*)

//stLocPos := stRelPos;
stLocPos := F_Add3DPoints(stRelPos,F_Add3DPoints(stLocPos,stCamOffsetMarker1));
stLocPos.Z := stLocPos.Z + stDimension.Height + rZOffset;
CASE eTargetRef OF
	E_TargetRef.TARGETREF_LeftBottom:
		;
	E_TargetRef.TARGETREF_LeftTop:
		stLocPos.Y := stLocPos.Y + stDimension.Depth ;
	E_TargetRef.TARGETREF_RightBottom:
		stLocPos.X := stLocPos.X + stDimension.Width;
	E_TargetRef.TARGETREF_RightTop:
		stLocPos.X := stLocPos.X + stDimension.Width;
		stLocPos.Y := stLocPos.Y + stDimension.Depth;
	E_TargetRef.TARGETREF_Center:
		stLocPos.X := stLocPos.X + stDimension.Width / 2.0;
		stLocPos.Y := stLocPos.Y + stDimension.Depth / 2.0;
		(*
	E_TargetRef.TARGETREF_SpecPoint:
		IF nNoOfSpecPoints = 2 THEN
			IF nParam1 = 1 THEN	//Mark1
				stLocPos := F_Add3DPoints(stLocPos,stMark1);
			ELSIF nParam1 = 2 THEN	//Mark2
				stLocPos := F_Add3DPoints(stLocPos,stMark2);
			ELSE
				nErrorId := E_ErrorIdCmd.ERRORID_InvalidTargetPointNr;
			END_IF	
		ELSE
			nErrorId := E_ErrorIdCmd.ERRORID_InvalidTargetPointNr;	
		END_IF*)
	
ELSE
	nErrorId := E_ErrorIdCmd.ERRORID_InvalidTargetPointRef;
END_CASE

IF nErrorId > 0 THEN
	RETURN;
END_IF


stLocPosAligned := stLocPos;


//Marker 1 Position wird noch nicht übermittelt von GUI. TODO: Wenn Übermittlung funktioniert, dann raus löschen
stMarker1Position.X := 4500;
stMarker1Position.Y := 4500;

IF rTargetRot <> 0 THEN	//Im Grunde müssten sich die Marken genauso drehen lassen
	//Offset
	//stLocPosAligned.X := stLocPosAligned.X - stCamOffsetMarker1.X;	
	//stLocPosAligned.Y := stLocPosAligned.Y - stCamOffsetMarker1.Y;
	//Drehen
	stLocPosAligned := F_RotatePoint(stLocPosAligned,F_Add3DPoints(stMarker1Position,stCamOffsetMarker1),rTargetRot/1000);
END_IF

//stLocPos := F_Add3DPoints(stLocPos,stRelPos);
//stLocPosAligned := F_Add3DPoints(stLocPosAligned,stRelPos);

IF pChildPos > 0 THEN
		lrAngle := rTargetRot/1000;
	//IF THIS^.rTargetRot <> 0 THEN
		pChildPos^ := F_RotatePoint(pChildPos^,stNull,rTargetRot/1000);
		//END_IF
		pChildPos^.X := pChildPos^.X + stLocPosAligned.X -stLocPos.X;
		pChildPos^.Y := pChildPos^.Y + stLocPosAligned.Y -stLocPos.Y;
	
	stLocPos.X := pChildPos^.X + stLocPos.X;
	stLocPos.Y := pChildPos^.Y + stLocPos.Y;
	stLocPos.Z := pChildPos^.Z + stLocPos.Z;
	(*ELSE
	pChildPos^.X := pChildPos^.X + stLocPosAligned.X - stLocPos.X;
	pChildPos^.Y := pChildPos^.Y + stLocPosAligned.Y - stLocPos.Y;

	stLocPos.X := pChildPos^.X + stLocPos.X;
	stLocPos.Y := pChildPos^.Y + stLocPos.Y;
	stLocPos.Z := pChildPos^.Z + stLocPos.Z;*)

	
	
ELSE
	stLocPos := stLocPosAligned;
END_IF

IF pParentTarget > 0 THEN
	IF pParentSlot > 0 THEN
 		stLocPos := pParentTarget^.M_GetAbsPos(pChildPos := ADR(stLocPos), eTargetRef:= E_TargetRef.TARGETREF_Slot,
													nParam1:= pParentSlot^.P_nNr,
													nParam2:= 0, nParam3:= 0,nZLevel:= 0,
													lrAngle => lrAngle, nErrorId=> nErrorId);
	ELSE
 		stLocPos := pParentTarget^.M_GetAbsPos(pChildPos := ADR(stLocPos), eTargetRef:= E_TargetRef.TARGETREF_LeftBottom,
													nParam1:= 0,
													nParam2:= 0, nParam3:= 0,nZLevel:= 0,
													lrAngle => lrAngle, nErrorId=> nErrorId);
	END_IF
END_IF

IF nErrorId > 0 THEN
	RETURN;
END_IF
(*
IF bIsAligned THEN
	lrAngle := lrAngle + THIS^.lrAngle;	
END_IF*)

M_GetAbsPos := stLocPos;
END_METHOD

METHOD M_GetAllProps : ERRORID
VAR_INPUT
	refCmdData : REFERENCE TO ST_CmdData;
END_VAR
SUPER^.M_GetAllProps(refCmdData); //wurde auskommentiert weil die Specific Points ein Relikt aus einer alten Version sind und nicht mehr gebraucht werden

//Alignment-Marken
	nCurrentPropIndex := 1;
	nCurrentPropIndex := nCurrentPropIndex + 1;
	refCmdData.n32Data[nCurrentPropIndex] := REAL_TO_DINT(stRelPos.X);				//2
	nCurrentPropIndex := nCurrentPropIndex + 1;                         			
	refCmdData.n32Data[nCurrentPropIndex] := REAL_TO_DINT(stRelPos.Y);				//3
	nCurrentPropIndex := nCurrentPropIndex + 1;                         			
	refCmdData.n32Data[nCurrentPropIndex] := REAL_TO_DINT(stRelPos.Z);				//4		
	nCurrentPropIndex := nCurrentPropIndex + 1;                                 	
	refCmdData.n32Data[nCurrentPropIndex] := REAL_TO_DINT(stDimension.Width);		//5
	nCurrentPropIndex := nCurrentPropIndex + 1;                                 	
	refCmdData.n32Data[nCurrentPropIndex] := REAL_TO_DINT(stDimension.Depth);		//6
	nCurrentPropIndex := nCurrentPropIndex + 1;                                 	
	refCmdData.n32Data[nCurrentPropIndex] := REAL_TO_DINT(stDimension.Height);		//7
	nCurrentPropIndex := nCurrentPropIndex + 1;                                 	
	refCmdData.n32Data[nCurrentPropIndex] := REAL_TO_DINT(rFreeHeight);				//8
	nCurrentPropIndex := nCurrentPropIndex + 1;                                 	
	refCmdData.n32Data[nCurrentPropIndex] := REAL_TO_DINT(rZOffset);				//9
	nCurrentPropIndex := nCurrentPropIndex + 1;                                 	
	refCmdData.n32Data[nCurrentPropIndex] := REAL_TO_DINT(stMarker1Position.X);		//10
	nCurrentPropIndex := nCurrentPropIndex + 1;
	refCmdData.n32Data[nCurrentPropIndex] := REAL_TO_DINT(stCamOffsetMarker1.X);	//11
	nCurrentPropIndex := nCurrentPropIndex + 1;
	refCmdData.n32Data[nCurrentPropIndex] := REAL_TO_DINT(stCamOffsetMarker1.Y);	//12
	nCurrentPropIndex := nCurrentPropIndex + 1;                                 
	refCmdData.n32Data[nCurrentPropIndex] := REAL_TO_DINT(stCamOffsetMarker1.Z);	//13
	nCurrentPropIndex := nCurrentPropIndex + 1;                                 
	refCmdData.n32Data[nCurrentPropIndex] := REAL_TO_DINT(rTargetRot);				//14
	nCurrentPropIndex := nCurrentPropIndex + 1;                                 
	refCmdData.n32Data[nCurrentPropIndex] := REAL_TO_DINT(stCamOffsetMarker2.X);	//15
(*
refCmdData.n32Data[nCurrentPropIndex] := nNoOfSpecPoints;
IF nNoOfSpecPoints = 2 THEN
	nCurrentPropIndex := nCurrentPropIndex + 1;
	refCmdData.n32Data[nCurrentPropIndex] := REAL_TO_DINT(stMark1.X);
	nCurrentPropIndex := nCurrentPropIndex + 1;
	refCmdData.n32Data[nCurrentPropIndex] := REAL_TO_DINT(stMark1.Y);
	nCurrentPropIndex := nCurrentPropIndex + 1;
	refCmdData.n32Data[nCurrentPropIndex] := REAL_TO_DINT(stMark1.Z);		
	nCurrentPropIndex := nCurrentPropIndex + 1;
	refCmdData.n32Data[nCurrentPropIndex] := REAL_TO_DINT(stMark2.X);
	nCurrentPropIndex := nCurrentPropIndex + 1;
	refCmdData.n32Data[nCurrentPropIndex] := REAL_TO_DINT(stMark2.Y);
	nCurrentPropIndex := nCurrentPropIndex + 1;
	refCmdData.n32Data[nCurrentPropIndex] := REAL_TO_DINT(stMark2.Z);		
END_IF
*)
END_METHOD

METHOD M_SetAllProps : ERRORID
VAR_INPUT
	refCmdData : REFERENCE TO  ST_CmdData;
END_VAR

VAR
	rTemp: REAL;
	bFlag: BOOL;
END_VAR
//Hier wird ausdrücklich nicht die Basisklasse aufgerufen, da nur hier gecheckt wird, ob sich die RelPos in XY und die Breite und
//Tiefe geändert haben um das Alignment zurückzusetzen.
nNoOfProps := 16;
//Relative Koordinaten
nCurrentPropIndex := 2;
rTemp := DINT_TO_REAL(refCmdData.n32Data[nCurrentPropIndex]);
IF rTemp <> stRelPos.X THEN
	stRelPos.X := rTemp;
	bFlag := TRUE;
END_IF
nCurrentPropIndex := nCurrentPropIndex + 1;	//3
rTemp := DINT_TO_REAL(refCmdData.n32Data[nCurrentPropIndex]);
IF rTemp <> stRelPos.Y THEN
	stRelPos.Y := rTemp;
	bFlag := TRUE;
END_IF
nCurrentPropIndex := nCurrentPropIndex + 1;	//4
rTemp := DINT_TO_REAL(refCmdData.n32Data[nCurrentPropIndex]);
IF rTemp <> stRelPos.Z THEN
	stRelPos.Z := rTemp;
	bFlag := TRUE;
END_IF

//Dimensionen
nCurrentPropIndex := nCurrentPropIndex + 1;	//5
rTemp := DINT_TO_REAL(refCmdData.n32Data[nCurrentPropIndex]);
IF rTemp <> stDimension.Width THEN
	stDimension.Width := rTemp;
	bFlag := TRUE;
END_IF
nCurrentPropIndex := nCurrentPropIndex + 1;	//6
rTemp := DINT_TO_REAL(refCmdData.n32Data[nCurrentPropIndex]);
IF rTemp <> stDimension.Depth THEN
	stDimension.Depth := rTemp;
	bFlag := TRUE;
END_IF
nCurrentPropIndex := nCurrentPropIndex + 1;	//7
rTemp := DINT_TO_REAL(refCmdData.n32Data[nCurrentPropIndex]);
IF rTemp <> stDimension.Height THEN
	stDimension.Height := rTemp;
	bFlag := TRUE;
END_IF
nCurrentPropIndex := nCurrentPropIndex + 1;	//8
rFreeHeight := DINT_TO_REAL(refCmdData.n32Data[nCurrentPropIndex]);

nCurrentPropIndex := nCurrentPropIndex + 1;	//9
rZOffset := DINT_TO_REAL(refCmdData.n32Data[nCurrentPropIndex]);
//nNoOfProps := nCurrentPropIndex + 3;

//Marker-Points
nCurrentPropIndex := nCurrentPropIndex + 1;	//10
rTemp := DINT_TO_REAL(refCmdData.n32Data[nCurrentPropIndex]);
IF rTemp <> stMarker1Position.X THEN
	stMarker1Position.X := rTemp;
	bFlag := TRUE;
END_IF

nCurrentPropIndex := nCurrentPropIndex + 1;	//11
rTemp := DINT_TO_REAL(refCmdData.n32Data[nCurrentPropIndex]);
IF rTemp <> stCamOffsetMarker1.X THEN
	stCamOffsetMarker1.X := rTemp;
	bFlag := TRUE;
END_IF

nCurrentPropIndex := nCurrentPropIndex + 1;	//12
rTemp := DINT_TO_REAL(refCmdData.n32Data[nCurrentPropIndex]);
IF rTemp <> stCamOffsetMarker1.Y THEN
	stCamOffsetMarker1.Y := rTemp;
	bFlag := TRUE;
END_IF

nCurrentPropIndex := nCurrentPropIndex + 1;	//13
rTemp := DINT_TO_REAL(refCmdData.n32Data[nCurrentPropIndex]);
IF rTemp <> stCamOffsetMarker1.Z THEN
	stCamOffsetMarker1.Z := rTemp;
	bFlag := TRUE;
END_IF

nCurrentPropIndex := nCurrentPropIndex + 1;	//14
rTemp := DINT_TO_REAL(refCmdData.n32Data[nCurrentPropIndex]);
IF rTemp <> rTargetRot THEN
	rTargetRot := rTemp;
	bFlag := TRUE;
END_IF

nCurrentPropIndex := nCurrentPropIndex + 1;	//15
rTemp := DINT_TO_REAL(refCmdData.n32Data[nCurrentPropIndex]);
IF rTemp <> stCamOffsetMarker2.X THEN
	stCamOffsetMarker2.X := rTemp;
	bFlag := TRUE;
END_IF
//Alignment-Marken
(*
nSpecPropIndex := nCurrentPropIndex;
nNoOfSpecPoints := DINT_TO_USINT(refCmdData.n32Data[nCurrentPropIndex]);
IF nNoOfSpecPoints = 0 THEN
	;
ELSIF nNoOfSpecPoints = 2 THEN
	//Wenn sich eine Position (X oder Y) geändert hat, dann Alignment-Flag zurücksetzen
	nCurrentPropIndex := nCurrentPropIndex + 1;
	rTemp := DINT_TO_REAL(refCmdData.n32Data[nCurrentPropIndex]);
	IF rTemp <> stMark1.X THEN
		stMark1.X := rTemp;
		bFlag := TRUE;
 	END_IF
	nCurrentPropIndex := nCurrentPropIndex + 1;
	rTemp := DINT_TO_REAL(refCmdData.n32Data[nCurrentPropIndex]);
	IF rTemp <> stMark1.Y THEN
		stMark1.Y := rTemp;
		bFlag := TRUE;
 	END_IF
	nCurrentPropIndex := nCurrentPropIndex + 1;
	stMark1.Z := DINT_TO_REAL(refCmdData.n32Data[nCurrentPropIndex]);
	nCurrentPropIndex := nCurrentPropIndex + 1;
	rTemp := DINT_TO_REAL(refCmdData.n32Data[nCurrentPropIndex]);
	IF rTemp <> stMark2.X THEN
		stMark2.X := rTemp;
		bFlag := TRUE;
 	END_IF
	nCurrentPropIndex := nCurrentPropIndex + 1;
	rTemp := DINT_TO_REAL(refCmdData.n32Data[nCurrentPropIndex]);
	IF rTemp <> stMark2.Y THEN
		stMark2.Y := rTemp;
		bFlag := TRUE;
 	END_IF
	nCurrentPropIndex := nCurrentPropIndex + 1;
	stMark2.Z := DINT_TO_REAL(refCmdData.n32Data[nCurrentPropIndex]);
	IF bFlag AND bIsAligned THEN
		bIsAligned := FALSE;
		lrAngle := 0.0;
	END_IF
ELSE
	M_SetAllProps := E_ErrorIdObjMgmt.ERRORID_InvalidNoOfSpecPoints;
END_IF
*)
P_pWorkplate^.P_bCalcCollisHeight := TRUE;
END_METHOD

METHOD M_SetMark1Act	//Auskommentiert, wird nicht mehr genutzt
VAR_INPUT
	///ist eine absolute Position
	stAbsPos: ST_3DPoint;
END_VAR
VAR
	stLeftBottom : ST_3DPoint;
	stNullPoint : ST_3DPoint;
	lrAngle : LREAL;
	bTempIsAligned : BOOL;
END_VAR
//Den aktuellen Wert der Marke 1 setzen
//Dieser bezieht sich auf die untere linke Ecke
//Bei einem erneutem Einteachen dürfte es eigentlich kein Problem auftauchen, da hier ja der eigene vorher schon berechnete Winkel
//noch nicht beachtet wird. Das könnte man bei einem Test mal beweisen
//doch, in der Methode M_GetAbsPos() wird die bestehende Korrektur schon mit berücksichtigt.
//es wäre gut, wenn die Methode noch einen Parameter hätte, der bewirkt, das die eigene Korrektur nicht berücksichtigt.
//warum nicht das bIsAligned mal kurzfristig zurücksetzen?
(*
bTempIsAligned := bIsAligned;
bIsAligned := FALSE;
stLeftBottom := M_GetAbsPos(0, E_TargetRef.TARGETREF_LeftBottom, 0, 0, 0, 0,lrAngle=>lrAngle);
bIsAligned := bTempIsAligned;
stMark1Act.X := stAbsPos.X - stLeftBottom.X;
stMark1Act.Y := stAbsPos.Y - stLeftBottom.Y;

//Falls das ParentTarget gedreht ist, dann muss diese Marke um den kumulierten Drehwinkel der Parents zurückgedreht werden
stMark1Act := F_RotatePoint(stMark1Act,stNullPoint,-lrAngle);*)
END_METHOD

METHOD M_SetMark2Act	//Auskommentiert, wird nicht mehr genutzt
VAR_INPUT
	///ist eine absolute Position
	stAbsPos: ST_3DPoint;
END_VAR
VAR
	stLeftBottom: ST_3DPoint;
	stNullPoint : ST_3DPoint;
	lrAngle : LREAL;
	bTempIsAligned : BOOL;
END_VAR
(*bTempIsAligned := bIsAligned;
bIsAligned := FALSE;
stLeftBottom := M_GetAbsPos(0, E_TargetRef.TARGETREF_LeftBottom, 0, 0, 0, 0,lrAngle=>lrAngle);
bIsAligned := bTempIsAligned;
stMark2Act.X := stAbsPos.X - stLeftBottom.X;
stMark2Act.Y := stAbsPos.Y - stLeftBottom.Y;
//Falls das ParentTarget gedreht ist, dann muss diese Marke um den kumulierten Drehwinkel der Parents zurückgedreht werden
stMark2Act := F_RotatePoint(stMark2Act,stNullPoint,-lrAngle);*)
END_METHOD

METHOD M_SetSingleProp : ERRORID
VAR_INPUT
	refCmdData: REFERENCE TO ST_CmdData;
END_VAR
VAR
	rTemp: REAL;
	bFlag: BOOL;
END_VAR
	//Hier wird die Basisklasse ausgelassen, da auf Änderung der RelPos und Dimensionen für das Rücksetzen des Alignments gecheckt wird.
	rTemp := DINT_TO_REAL(refCmdData.n32Data[0]);
	CASE refCmdData.aHeader[1] OF
		2:	//XPosRel
			IF rTemp <> stRelPos.X THEN
				stRelPos.X := rTemp;
				bFlag := TRUE; 	
			END_IF
		3:	//YPosRel
			IF rTemp <> stRelPos.Y THEN
				stRelPos.Y := rTemp;
				bFlag := TRUE; 	
			END_IF
		4:	//ZPosRel
			IF rTemp <> stRelPos.Z THEN
				stRelPos.Z := rTemp;
				bFlag := TRUE;
				P_pWorkplate^.P_bCalcCollisHeight := TRUE; 	
			END_IF
		5:	//Width
			IF rTemp <> stDimension.Width THEN
				stDimension.Width := rTemp;
				bFlag := TRUE;
			END_IF
		6:	//Depth
			IF rTemp <> stDimension.Depth THEN
				stDimension.Depth := rTemp;
				bFlag := TRUE;
			END_IF
		7:	//Height
			IF rTemp <> stDimension.Height THEN
				stDimension.Height := rTemp;
				bFlag := TRUE;
				P_pWorkplate^.P_bCalcCollisHeight := TRUE; 	
			END_IF
		8:	//FreeHeight
			IF rTemp <> rZOffset THEN
				rZOffset := rTemp;
				bFlag := TRUE; 	
			END_IF
		9:	//ZOffset
			IF rTemp <> rFreeHeight THEN
				rFreeHeight := rTemp;
				bFlag := TRUE; 	
			END_IF
		10:	//Marker1Position.X
			IF rTemp <> stMarker1Position.X THEN
				stMarker1Position.X := rTemp;
				bFlag := TRUE; 	
			END_IF
		11:	//stCamOffsetMarker1.X
			IF rTemp <> stCamOffsetMarker1.X THEN
				stCamOffsetMarker1.X := rTemp;
				bFlag := TRUE; 	
			END_IF
		12:	//stCamOffsetMarker1.Y
			IF rTemp <> stCamOffsetMarker1.Y THEN
				stCamOffsetMarker1.Y := rTemp;
				bFlag := TRUE; 	
			END_IF		
		13:	//stCamOffsetMarker1.Z
			IF rTemp <> stCamOffsetMarker1.Z THEN
				stCamOffsetMarker1.Z := rTemp;
				bFlag := TRUE; 	
			END_IF
		14:	//rTargetRot
			 IF rTemp <> rTargetRot THEN
				rTargetRot := rTemp;
				bFlag := TRUE; 	
			END_IF
		15:	//stCamOffsetMarker2.X
			 IF rTemp <> stCamOffsetMarker2.X THEN
				stCamOffsetMarker2.X := rTemp;
				bFlag := TRUE; 	
			END_IF
	END_CASE
(*	IF bFlag AND bIsAligned THEN
		bIsAligned := FALSE;
		lrAngle := 0.0;
	END_IF	
ELSE
	IF (nSpecPropIndex + 1) = refCmdData.aHeader[1] THEN
		rZOffset := DINT_TO_REAL(refCmdData.n32Data[0]);
	ELSE
		M_SetSingleProp := SUPER^.M_SetSingleProp(refCmdData);
	END_IF	
END_IF*)
END_METHOD

PROPERTY P_bIsAligned : BOOL
GET
//P_bIsAligned := bIsAligned;
END_GET
SET
//bIsAligned := P_bIsAligned;
END_SET
END_PROPERTY

PROPERTY P_lrAbsAngle : LREAL
GET
IF pParentTarget > 0 THEN
	P_lrAbsAngle := pParentTarget^.P_lrAbsAngle + rTargetRot/1000;
END_IF
END_GET
END_PROPERTY

PROPERTY P_lrAngle : LREAL
GET
P_lrAngle := rTargetRot/1000;
END_GET
SET
rTargetRot := P_lrAngle*1000;
END_SET
END_PROPERTY

PROPERTY P_rOffsetX : REAL
GET
(*IF bIsAligned THEN
	P_rOffsetX := stMark1Act.X - stMark1.X;
END_IF*)
END_GET
END_PROPERTY

PROPERTY P_rOffsetY : REAL
GET
(*IF bIsAligned THEN
	P_rOffsetY := stMark1Act.Y - stMark1.Y;
END_IF*)
END_GET
END_PROPERTY

PROPERTY P_stMark1 : ST_3DPoint
GET
//P_stMark1 := F_Add3DPoints(stMark1,P_stAbsPosLB);
END_GET
END_PROPERTY

END_FUNCTION_BLOCK

// ---- Objects/Targets/Passive/FB_SpotArray.TcPOU
{attribute 'enable_dynamic_creation'}
FUNCTION_BLOCK FB_SpotArray EXTENDS FB_Array
VAR_INPUT
END_VAR
VAR_OUTPUT
END_VAR
VAR
END_VAR

METHOD FB_init : BOOL
VAR_INPUT
	bInitRetains : BOOL; // if TRUE, the retain variables are initialized (warm start / cold start)
	bInCopyCode : BOOL;  // if TRUE, the instance afterwards gets moved into the copy code (online change)
END_VAR
eObjectType := E_ObjectType.OBJECTTYPE_SpotArray;
eObjectGroup := E_ObjectGroup.OBJECTGROUP_Target OR E_ObjectGroup.OBJECTGROUP_Array;
END_METHOD

METHOD M_AddChild : ERRORID
VAR_INPUT
	pObject : POINTER TO FB_Object;
	nSlotNr	: UINT;
	nIndex 	: INT;
END_VAR
//Kann folgende Objekte aufnehmen:
IF pObject > 0 THEN
	IF pObject^.P_eObjectType = E_ObjectType.OBJECTTYPE_Point THEN
		M_AddChild := SUPER^.M_AddChild(pObject,nSlotNr,nIndex);
	ELSE
		M_AddChild := E_ErrorIdObjMgmt.ERRORID_InvalidParentObject;
	END_IF
ELSE
	M_AddChild := E_ErrorIdObjMgmt.ERRORID_InvalidParentObject;
END_IF
END_METHOD

END_FUNCTION_BLOCK

// ---- Objects/Pieces/FB_Stamp.TcPOU
{attribute 'enable_dynamic_creation'}
FUNCTION_BLOCK FB_Stamp EXTENDS FB_PieceBase
VAR_INPUT
END_VAR
VAR_OUTPUT
END_VAR
VAR
END_VAR

METHOD FB_init : BOOL
VAR_INPUT
	bInitRetains : BOOL; // if TRUE, the retain variables are initialized (warm start / cold start)
	bInCopyCode : BOOL;  // if TRUE, the instance afterwards gets moved into the copy code (online change)
END_VAR
eObjectType := E_ObjectType.OBJECTTYPE_Stamp;
eObjectGroup := E_ObjectGroup.OBJECTGROUP_Piece;
END_METHOD

END_FUNCTION_BLOCK

// ---- Objects/Pieces/FB_Tip.TcPOU
{attribute 'enable_dynamic_creation'}
FUNCTION_BLOCK FB_Tip EXTENDS FB_UsingPiece
VAR_INPUT
END_VAR
VAR_OUTPUT
END_VAR
VAR
END_VAR

METHOD FB_init : BOOL
VAR_INPUT
	bInitRetains : BOOL; // if TRUE, the retain variables are initialized (warm start / cold start)
	bInCopyCode : BOOL;  // if TRUE, the instance afterwards gets moved into the copy code (online change)
END_VAR
bUsingPiece := TRUE;
eObjectType := E_ObjectType.OBJECTTYPE_Tip;
eObjectGroup := E_ObjectGroup.OBJECTGROUP_Piece;
END_METHOD

END_FUNCTION_BLOCK

// ---- Objects/Targets/Passive/FB_TargetTray.TcPOU
{attribute 'enable_dynamic_creation'}
FUNCTION_BLOCK FB_TargetTray EXTENDS FB_SlotTarget
VAR_INPUT
END_VAR
VAR_OUTPUT
END_VAR
VAR
END_VAR

METHOD FB_init : BOOL
VAR_INPUT
	bInitRetains : BOOL; // if TRUE, the retain variables are initialized (warm start / cold start)
	bInCopyCode : BOOL;  // if TRUE, the instance afterwards gets moved into the copy code (online change)
END_VAR
eObjectType := E_ObjectType.OBJECTTYPE_TargetTray;
eObjectGroup := E_ObjectGroup.OBJECTGROUP_Target;
END_METHOD

METHOD M_AddChild : ERRORID
VAR_INPUT
	pObject : POINTER TO FB_Object;
	nSlotNr	: UINT;
	nIndex 	: INT;
END_VAR
//Kann alle Targets aufnehmen
IF pObject > 0 THEN
	IF pObject^.M_bIsGroup(E_ObjectGroup.OBJECTGROUP_Target) THEN
		M_AddChild := SUPER^.M_AddChild(pObject,nSlotNr,nIndex);
	ELSE
		M_AddChild := E_ErrorIdObjMgmt.ERRORID_InvalidParentObject;
	END_IF
ELSE
	M_AddChild := E_ErrorIdObjMgmt.ERRORID_InvalidParentObject;
END_IF
END_METHOD

END_FUNCTION_BLOCK

// ---- Objects/Pieces/FB_VialClosed.TcPOU
{attribute 'enable_dynamic_creation'}
FUNCTION_BLOCK FB_VialClosed EXTENDS FB_Vial
VAR_INPUT
END_VAR
VAR_OUTPUT
END_VAR
VAR
END_VAR

{attribute 'object_name' := 'FB_init'}
METHOD FB_init : BOOL
VAR_INPUT
	/// if TRUE, the retain variables are initialized (warm start / cold start)
	bInitRetains: BOOL;
	/// if TRUE, the instance afterwards gets moved into the copy code (online change)
	bInCopyCode: BOOL;
END_VAR
eObjectType := E_ObjectType.OBJECTTYPE_VialClosed;
END_METHOD

END_FUNCTION_BLOCK

// ---- Objects/Targets/Passive/FB_CleaningBrush.TcPOU
{attribute 'enable_dynamic_creation'}
FUNCTION_BLOCK FB_CleaningBrush EXTENDS FB_TargetBase
VAR_INPUT
END_VAR
VAR_OUTPUT
END_VAR

VAR
	rMargin  : REAL;
END_VAR

METHOD FB_init : BOOL
VAR_INPUT
	bInitRetains : BOOL; // if TRUE, the retain variables are initialized (warm start / cold start)
	bInCopyCode : BOOL;  // if TRUE, the instance afterwards gets moved into the copy code (online change)
END_VAR
eObjectType := E_ObjectType.OBJECTTYPE_CleaningBrush;
eObjectGroup := E_ObjectGroup.OBJECTGROUP_Target;
END_METHOD

METHOD M_GetAllProps : ERRORID
VAR_INPUT
	refCmdData : REFERENCE TO  ST_CmdData;
END_VAR
SUPER^.M_GetAllProps(refCmdData);
nCurrentPropIndex := nCurrentPropIndex + 1;
refCmdData.n32Data[nCurrentPropIndex] := REAL_TO_DINT(rMargin);
END_METHOD

{attribute 'object_name' := 'M_SetAllProps'}
METHOD M_SetAllProps : ERRORID
VAR_INPUT
	refCmdData	: REFERENCE TO ST_CmdData;
END_VAR
M_SetAllProps := SUPER^.M_SetAllProps(refCmdData);

IF M_SetAllProps > 0 THEN
	RETURN;
END_IF

nCurrentPropIndex := nCurrentPropIndex + 1;
rMargin := DINT_TO_REAL(refCmdData.n32Data[nCurrentPropIndex]);
nNoOfProps := nCurrentPropIndex + 1;
END_METHOD

PROPERTY P_rMargin : REAL
GET
P_rMargin := rMargin;
END_GET
END_PROPERTY

END_FUNCTION_BLOCK

// ---- Objects/Tools/FB_PowderPip.TcPOU
FUNCTION_BLOCK FB_PowderPip EXTENDS FB_GCodeTool

VAR

	//Specproperties
	pPneuChannelPress	: POINTER TO FB_PneuChannelRef;
	pPneuChannelVac		: POINTER TO FB_PneuChannelRef;
	
	nDOutChanValvePress	: USINT;	//Digitaler Ausgangskanal MzHead Druckventil
	nDOutChanValveVac	: USINT;	//Digitaler Ausgangskanal MzHead Vakuumventil 
	
	//****************************************Aktionvariablen****************************************************
	
	//Action: "InitTool"
	bInitTool			: BOOL;
	nStateA_InitTool	: USINT;	

	//Action: "SetPressure"
	bSetPress			: BOOL;
	fbSetPress			: FB_SetPressure;

	//Action: "SetVacuum"
	bSetVacuum			: BOOL;
	fbSetVacuum			: FB_SetPressure;
	
	//Action: "SwitchPressure"
	bSwitchPress		: BOOL;
	nStateA_SwitchPress	: USINT;	//State von A_SwitchPress()
	ePressCtrl			: E_PressCtrl;
	eCurrPressCtrl 		: E_PressCtrl; 
	tPressTime			: TIME;		//Öffnungszeit Druckventil
	timerPress			: TON;		//Timer für Öffnungszeit Druckventil
	
	//Action: "PulsePressure"
	bPulsePress			: BOOL;
	nStateA_PulsePress	: USINT;	//State von A_PulsePress()
	eSwitchCtrlPhase1	: E_PressCtrl;		//
	eSwitchCtrlPhase2	: E_PressCtrl;		//
	nPulseDutycycle		: UINT;		//Tastverhältnis (0-100%)
	nTimePhase1			: UINT;
	nTimePhase2			: UINT;
	timerPulse			: TON;		//Timer
	nSetpointPulses		: UINT;		//Soll Anzahl an Pulses
	nCurrentPulses		: UINT;		//aktuelle Anzahl an Pulses
	bPulseOn			: BOOL;	
	
	//Action: "PickPut
	bPickPut			: BOOL;
	nStateA_PickPut		: USINT;
	ePickPutMode		: E_PickPutMode;
	nIntakeVac			: INT;
	tIntakeTime			: TIME;
	nHoldVac			: INT;
	nBlowOutPress		: INT;
	nBlowOutPulseTime	: UINT;
	nBlowOutPulses		: UINT;
	timerPickPut		: TON;
	stActionDataPickPut	: ST_ActionData;	
	
END_VAR

IF eCurrentState = E_MachineState.MACHINESTATE_Active THEN
	
	IF bInitTool THEN
		A_InitTool();
		IF nStateA_InitTool >= 80 THEN
			IF nStateA_InitTool >= 99 THEN
				bError := TRUE;
			END_IF
			bInitTool := FALSE;
			nStateA_InitTool := 0;
			M_RemoveListEntry(nSearchValue:= E_Action.ACTION_Init);
		END_IF		
	END_IF
	
	IF bPickPut THEN
		A_PickPut();
		IF nStateA_PickPut >= 80 THEN
			IF nStateA_PickPut >= 99 THEN
				bError := TRUE;
			END_IF
			bPickPut := FALSE;
			nStateA_PickPut := 0;
			M_RemoveListEntry(nSearchValue:= E_Action.ACTION_PickPutPowder);
		END_IF
	END_IF		
	
	IF bSetPress THEN
		fbSetPress(pPneuChannelRef:= pPneuChannelPress);
		IF NOT fbSetPress.bBusy THEN
			IF fbSetPress.bError THEN
				bError := TRUE;
				stError.ErrorId := fbSetPress.nErrorId;
				stError.POU := E_POU.POU_FB_PowderPip;
				fbErrorList.M_Add(stError);
			END_IF
			bSetPress := FALSE;
			fbSetPress(pPneuChannelRef:= pPneuChannelPress, bExecute:= FALSE);
			M_RemoveListEntry(nSearchValue:= E_Action.ACTION_SetPressure);
		END_IF
	END_IF	

	IF bSetVacuum THEN
		fbSetVacuum(pPneuChannelRef:= pPneuChannelVac);
		IF NOT fbSetVacuum.bBusy THEN
			IF fbSetVacuum.bError THEN
				bError := TRUE;
				stError.ErrorId := fbSetVacuum.nErrorId;
				stError.POU := E_POU.POU_FB_PowderPip;
				fbErrorList.M_Add(stError);
			END_IF
			bSetVacuum := FALSE;
			fbSetVacuum(pPneuChannelRef:= pPneuChannelVac, bExecute:= FALSE);
			M_RemoveListEntry(nSearchValue:= E_Action.ACTION_SetVacuum);
		END_IF
	END_IF	

	IF bSwitchPress THEN	//Druck/Vakuum Ein/Aus
		A_SwitchPress();
		IF nStateA_SwitchPress >= 80 THEN
			IF nStateA_SwitchPress >= 99 THEN
				bError := TRUE;
			END_IF
			bSwitchPress := FALSE;
			nStateA_SwitchPress := 0;
			M_RemoveListEntry(nSearchValue:= E_Action.ACTION_SwitchPressure);
		END_IF
	END_IF
	
	IF bPulsePress THEN
		A_PulsePress();
		IF nStateA_PulsePress >= 80 THEN
			IF nStateA_PulsePress >= 99 THEN
				bError := TRUE;
			END_IF
			bPulsePress := FALSE;
			nStateA_PulsePress := 0;
			M_RemoveListEntry(nSearchValue:= E_Action.ACTION_PulsePressure);
		END_IF
	END_IF
END_IF

SUPER^();	//FB_MzTool aufrufen

//Prozessdaten aktualisieren

IF pPneuChannelPress > 0 THEN
	stProcessData.n32Data[7] := pPneuChannelPress^.P_nCurrentPressure;
	stProcessData.n32Data[8] := pPneuChannelPress^.P_nCurrentPressure;
END_IF

IF pPneuChannelVac > 0 THEN
	stProcessData.n32Data[9] := pPneuChannelVac^.P_nSetPressure;
	stProcessData.n32Data[10] := pPneuChannelVac^.P_nCurrentPressure;
END_IF

IF pZAxisRef > 0 THEN
	IF pZAxisRef^.stOutput.nToolCtrl = 0 THEN
		stProcessData.n32Data[11] := E_PressCtrl.PRESSCTRL_Off;
	ELSIF pZAxisRef^.stOutput.nToolCtrl = 5 THEN
		stProcessData.n32Data[11] := E_PressCtrl.PRESSCTRL_PressOn;
	ELSIF pZAxisRef^.stOutput.nToolCtrl = 3 THEN
		stProcessData.n32Data[11] := E_PressCtrl.PRESSCTRL_VacOn;
	ELSE
		stProcessData.n32Data[11] := E_PressCtrl.PRESSCTRL_UNDEFINED;
	END_IF
END_IF

aObjProcData[nNotifyId] := stProcessData;

ACTION A_InitTool:
IF nStateA_InitTool = 0 THEN
	IF nDOutChanValvePress > 0 THEN
		pFbMultiZ^.aDigiOut[nDOutChanValvePress] := TRUE;	
	END_IF
	IF nDOutChanValveVac > 0 THEN
		pFbMultiZ^.aDigiOut[nDOutChanValveVac] := TRUE;	
	END_IF
	bInitToolOk := TRUE;
	nStateA_InitTool := 80;
END_IF
END_ACTION

ACTION A_PickPut:
CASE nStateA_PickPut OF
	0:	//Ventile schließen
		pZAxisRef^.stOutput.nToolCtrl := 0;
		//Wenn Pick IntakeVac einstellen, bei Put BlowOutPress einstellen
		MEMSET(ADR(stActionDataPickPut),0,SIZEOF(stActionDataPickPut));
		IF ePickPutMode = E_PickPutMode.MODE_Pick THEN
			stActionDataPickPut.eAction := E_Action.ACTION_SetVacuum;
			stActionDataPickPut.aParams[2] := nIntakeVac;	
		ELSIF ePickPutMode = E_PickPutMode.MODE_Put THEN
			stActionDataPickPut.eAction := E_Action.ACTION_SetPressure;
			stActionDataPickPut.aParams[2] := nBlowOutPress;
			GVL_HwRefIO.bTrigger1 := TRUE;
		END_IF
		stActionDataPickPut.aParams[1] := 1;	//Fertigmeldung erst, wenn Druck erreicht
		stActionDataPickPut.aParams[3] := 8;	//Tolerance +
		stActionDataPickPut.aParams[4] := 8;	//Tolerance -
		stActionDataPickPut.aParams[5] := 10000; //Timeout
		M_ExeAction(stActionDataPickPut);
		stActionDataPickPut.eAction := E_Action.ACTION_SwitchPressure;
		stActionDataPickPut.aParams[1] := E_PressCtrl.PRESSCTRL_Off;
		M_ExeAction(stActionDataPickPut);
		nStateA_PickPut := 1;
	
	1:	//Warten bis SollDruck erreioht ist
		IF NOT M_GetActionBusy(E_Action.ACTION_SetPressure) AND NOT M_GetActionBusy(E_Action.ACTION_SetVacuum)THEN
			IF ePickPutMode = E_PickPutMode.MODE_Pick THEN
				nStateA_PickPut := 2;
			ELSE
				nStateA_PickPut := 20;
			END_IF
		END_IF
		
	2:	//Pick - Switch Vacuum
		MEMSET(ADR(stActionDataPickPut),0,SIZEOF(stActionDataPickPut));
		stActionDataPickPut.eAction := E_Action.ACTION_SwitchPressure;
		stActionDataPickPut.aParams[1] := E_PressCtrl.PRESSCTRL_VacOn;
		stActionDataPickPut.aParams[2] := 0;
		M_ExeAction(stActionDataPickPut);
		timerPickPut(IN:=TRUE, PT:= tIntakeTime);
		nStateA_PickPut := 3;

	3:	//Warten, bis Zeit abgelaufen
		timerPickPut();
		IF timerPickPut.Q THEN
			timerPickPut(IN:= FALSE);
			MEMSET(ADR(stActionDataPickPut),0,SIZEOF(stActionDataPickPut));
			//HoldVac einstellen (wenn HoldVac = 0, dann SwitchPress auf Off
			IF nHoldVac < 0 THEN
				stActionDataPickPut.eAction := E_Action.ACTION_SetVacuum;
				stActionDataPickPut.aParams[1] := 0; //Ohne Überwachung
				stActionDataPickPut.aParams[2] := nHoldVac;
				M_ExeAction(stActionDataPickPut);
			ELSE
				stActionDataPickPut.eAction := E_Action.ACTION_SwitchPressure;
				stActionDataPickPut.aParams[1] := E_PressCtrl.PRESSCTRL_Off;
				stActionDataPickPut.aParams[2] := 0;
				M_ExeAction(stActionDataPickPut);
			END_IF
			nStateA_PickPut := 80;
		END_IF
		
	20:	//Put
		//PulsePressure
		MEMSET(ADR(stActionDataPickPut),0,SIZEOF(stActionDataPickPut));
		stActionDataPickPut.eAction := E_Action.ACTION_PulsePressure;
		stActionDataPickPut.aParams[1] := E_PressCtrl.PRESSCTRL_PressOn;
		stActionDataPickPut.aParams[2] := E_PressCtrl.PRESSCTRL_Off;
		stActionDataPickPut.aParams[3] := nBlowOutPulseTime * 2; //Periode
		stActionDataPickPut.aParams[4] := 50; //Dutycycle
		stActionDataPickPut.aParams[5] := nBlowOutPulses;
		stActionDataPickPut.aParams[6] := 1; //On
		M_ExeAction(stActionDataPickPut);
		nStateA_PickPut := 21;
		
	21: //Warten, bis Pulsen fertig
		IF NOT M_GetActionBusy(E_Action.ACTION_PulsePressure) THEN
			GVL_HwRefIO.bTrigger1 := FALSE;
			nStateA_PickPut := 80;
		END_IF
	
	70: //Abbrechen
		M_CancelAction(E_Action.ACTION_PulsePressure);
		stActionDataPickPut.eAction := E_Action.ACTION_SwitchPressure;
		stActionDataPickPut.aParams[1] := E_PressCtrl.PRESSCTRL_Off;
		M_ExeAction(stActionDataPickPut);
		timerPickPut(IN:= FALSE);
		nStateA_PickPut := 80;
		
END_CASE
END_ACTION

ACTION A_PulsePress:
CASE nStateA_PulsePress OF
	0:	//Phase1
		
		IF eSwitchCtrlPhase1 = E_PressCtrl.PRESSCTRL_Off THEN
			pZAxisRef^.stOutput.nToolCtrl := 0;
		ELSIF eSwitchCtrlPhase1 = E_PressCtrl.PRESSCTRL_PressOn THEN
			pZAxisRef^.stOutput.nToolCtrl := 5;
		ELSIF eSwitchCtrlPhase1 = E_PressCtrl.PRESSCTRL_VacOn THEN
			pZAxisRef^.stOutput.nToolCtrl := 3;
		END_IF

		timerPulse(IN:= TRUE, PT:= UINT_TO_TIME(nTimePhase1));
		IF timerPulse.Q THEN
			timerPulse(IN:= FALSE);
			nStateA_PulsePress := 1;
			nCurrentPulses := nCurrentPulses + 1;
		END_IF

	1:	//Phase2

		IF eSwitchCtrlPhase2 = E_PressCtrl.PRESSCTRL_Off THEN
			pZAxisRef^.stOutput.nToolCtrl := 0;
		ELSIF eSwitchCtrlPhase2 = E_PressCtrl.PRESSCTRL_PressOn THEN
			pZAxisRef^.stOutput.nToolCtrl := 5;
		ELSIF eSwitchCtrlPhase2 = E_PressCtrl.PRESSCTRL_VacOn THEN
			pZAxisRef^.stOutput.nToolCtrl := 3;
		END_IF

		timerPulse(IN:= TRUE, PT:= UINT_TO_TIME(nTimePhase2));
		IF timerPulse.Q THEN
			timerPulse(IN:= FALSE);
			IF nCurrentPulses = nSetpointPulses THEN
				pZAxisRef^.stOutput.nToolCtrl := 0;
				nStateA_PulsePress := 80;
			ELSIF nSetpointPulses = 0 AND NOT bPulseOn THEN
				pZAxisRef^.stOutput.nToolCtrl := 0;
				nStateA_PulsePress := 80;
			ELSE
				nStateA_PulsePress := 0;	
			END_IF
		END_IF
		
	70:	//Abbrechen
		timerPulse(IN:= FALSE);
		pZAxisRef^.stOutput.nToolCtrl := 0;
		nStateA_PulsePress := 80;
		
END_CASE
END_ACTION

ACTION A_Reset:
//Ist noch eine Aktion aktiv?
IF nStateA_ResetSpec = 0 THEN 
	IF bSetPress THEN
		bSetPress := FALSE;
		fbSetPress(bExecute:= FALSE, pPneuChannelRef:= pPneuChannelPress);
	END_IF

	IF bSetVacuum THEN
		bSetVacuum := FALSE;
		fbSetVacuum(bExecute:= FALSE, pPneuChannelRef:= pPneuChannelVac);
	END_IF
	
	IF bSwitchPress THEN 
		bSwitchPress := FALSE;
		nStateA_SwitchPress := 0;
	END_IF
	
	IF bPulsePress THEN
		bPulsePress := FALSE;
		nStateA_PulsePress := 0;
	END_IF
	
	IF bPickPut THEN
		bPickPut := FALSE;
		nStateA_PickPut := 0;
	END_IF
	
	nStateA_ResetSpec := 80;
END_IF

SUPER^.A_Reset();
END_ACTION

ACTION A_Stop:
IF nStateA_Stop = 0 THEN

	IF bSetPress THEN
		fbSetPress(bExecute:= FALSE, pPneuChannelRef:= pPneuChannelPress);
	END_IF

	IF bSetVacuum THEN
		fbSetVacuum(bExecute:= FALSE, pPneuChannelRef:= pPneuChannelVac);
	END_IF

	IF bSwitchPress AND nStateA_SwitchPress < 70 THEN
		nStateA_SwitchPress := 70;
	END_IF
	
	IF bPulsePress AND nStateA_PulsePress < 70 THEN
		nStateA_PulsePress := 70;
	END_IF
	
	IF bPickPut AND nStateA_PickPut < 70 THEN
		nStateA_PickPut := 70;
	END_IF

	nStateA_Stop := 1;
END_IF

SUPER^.A_Stop();
END_ACTION

ACTION A_SwitchPress:
// In jedem Zustand sollte umgeschalten werden
CASE nStateA_SwitchPress OF
	0:	//Wie soll geschalten werden?
		IF ePressCtrl = E_PressCtrl.PRESSCTRL_Off THEN
			eCurrPressCtrl := E_PressCtrl.PRESSCTRL_Off;
			pZAxisRef^.stOutput.nToolCtrl := 0;
			timerPress(IN:= FALSE);
			nStateA_SwitchPress := 80;
			RETURN;
		ELSIF ePressCtrl = E_PressCtrl.PRESSCTRL_PressOn THEN
			eCurrPressCtrl := E_PressCtrl.PRESSCTRL_PressOn;
			pZAxisRef^.stOutput.nToolCtrl := 5;
		ELSIF ePressCtrl = E_PressCtrl.PRESSCTRL_VacOn THEN
			eCurrPressCtrl := E_PressCtrl.PRESSCTRL_VacOn;
			pZAxisRef^.stOutput.nToolCtrl := 3;
		END_IF

		IF tPressTime > T#0MS THEN
			timerPress(IN:= TRUE, PT:= tPressTime);
			nStateA_SwitchPress := 1;
		ELSE
			nStateA_SwitchPress := 80;
		END_IF
		
	1:	//Timer
		//Haben sich die Eingangsparameter geändert?
		IF ePressCtrl <> eCurrPressCtrl THEN
			nStateA_SwitchPress := 0;
			timerPress(IN:= FALSE);
		END_IF
		timerPress();
		IF timerPress.Q THEN
			timerPress(IN:= FALSE);
			pZAxisRef^.stOutput.nToolCtrl := 0;
			eCurrPressCtrl := E_PressCtrl.PRESSCTRL_Off;
			nStateA_SwitchPress := 80;
		END_IF

	70:	//Abbrechen
		pZAxisRef^.stOutput.nToolCtrl := 0;
		timerPress(IN:= FALSE);
		nStateA_SwitchPress := 80;
		
	80:	//Haben sich die Eingangsparameter geändert?
		IF ePressCtrl <> eCurrPressCtrl THEN
			nStateA_SwitchPress := 0;
		END_IF
END_CASE
END_ACTION

METHOD FB_init : BOOL
VAR_INPUT
	bInitRetains : BOOL; // if TRUE, the retain variables are initialized (warm start / cold start)
	bInCopyCode : BOOL;  // if TRUE, the instance afterwards gets moved into the copy code (online change)
END_VAR
eObjectType := E_ObjectType.OBJECTTYPE_PowderPip;
eObjectGroup := E_ObjectGroup.OBJECTGROUP_MzTool OR E_ObjectGroup.OBJECTGROUP_Device;
END_METHOD

METHOD M_AddChild : ERRORID
VAR_INPUT
	pObject : POINTER TO FB_Object;
	nSlotNr	: UINT;
	nIndex 	: INT;
END_VAR
//Kann folgende Objekt-Typen aufnehmen
//Nozzle
IF pObject > 0 THEN
	IF pObject^.P_eObjectType = E_ObjectType.OBJECTTYPE_Nozzle THEN
		M_AddChild := SUPER^.M_AddChild(pObject,nSlotNr,nIndex);
	ELSE
		M_AddChild := E_ErrorIdObjMgmt.ERRORID_InvalidParentObject;
	END_IF
ELSE
	M_AddChild := E_ErrorIdObjMgmt.ERRORID_InvalidParentObject;
END_IF
END_METHOD

METHOD M_CancelAction
VAR_INPUT
	eAction : E_Action;
END_VAR
CASE eAction OF
	E_Action.ACTION_SetPressure:
		IF bSetPress THEN
			fbSetPress(bExecute:= FALSE, pPneuChannelRef:= pPneuChannelPress);
		END_IF
	
	E_Action.ACTION_SetVacuum:
		IF bSetVacuum THEN
			fbSetVacuum(bExecute:= FALSE, pPneuChannelRef:= pPneuChannelVac);
		END_IF

	E_Action.ACTION_SwitchPressure:
		IF bSwitchPress AND nStateA_SwitchPress < 70 THEN
			nStateA_SwitchPress := 70;
		END_IF

	E_Action.ACTION_PickPutPowder:
		IF bPickPut AND nStateA_PickPut < 70 THEN
			nStateA_PickPut := 70;
		END_IF

	E_Action.ACTION_PulsePressure:
		IF bPulsePress AND nStateA_PulsePress < 70 THEN
			nStateA_PulsePress := 70;
		END_IF	
ELSE
	SUPER^.M_CancelAction(eAction);
END_CASE
END_METHOD

METHOD M_CheckAction : ERRORID
VAR_INPUT
	refActionData 	: REFERENCE TO ST_ActionData;
	pCorrelObject	: POINTER TO FB_Object;
END_VAR
IF refActionData.eAction = E_Action.ACTION_MeasureTool THEN
	IF fbObjectDirectory.M_GetObjType(refActionData.nTarget) <> E_ObjectType.OBJECTTYPE_TipCalibrator THEN
		M_CheckAction := E_ErrorIdCmd.ERRORID_UnsuitableTarget;
	END_IF
ELSE
	M_CheckAction := SUPER^.M_CheckAction(refActionData, pCorrelObject);
END_IF
END_METHOD

METHOD M_ExeAction : ERRORID
VAR_INPUT
	refActionData : REFERENCE TO ST_ActionData;	
END_VAR
IF NOT (eCurrentState = E_MachineState.MACHINESTATE_Idle OR
	eCurrentState = E_MachineState.MACHINESTATE_Active OR
	eCurrentState = E_MachineState.MACHINESTATE_Ready) THEN
	M_ExeAction := E_ErrorIdCmd.ERRORID_InvalidState;
	RETURN;
END_IF

CASE refActionData.eAction OF
	
	E_Action.ACTION_Init:
		IF NOT bInitAxis AND NOT bInitTool THEN
			bInitAxis := TRUE;
			bInitTool := TRUE;
			fbList.A_AddHeadValue( hList := hList, putValue := E_Action.ACTION_Init);	//InitBase
			fbList.A_AddHeadValue( hList := hList, putValue := E_Action.ACTION_Init);	//InitSpec
		ELSE
			RETURN;
		END_IF		

	E_Action.ACTION_SetPressure:
		fbSetPress(bExecute:= FALSE, pPneuChannelRef:= pPneuChannelPress); //eventueller Fehler wird auch zurückgesetzt
		fbSetPress.bAwait := DINT_TO_BOOL(refActionData.aParams[1]);
		fbSetPress.nValue := DINT_TO_INT(refActionData.aParams[2]);
		fbSetPress.nTolerancePlus := DINT_TO_INT(refActionData.aParams[3]);
		fbSetPress.nToleranceMinus := DINT_TO_INT(refActionData.aParams[4]);
		fbSetPress.tTimeout := DINT_TO_TIME(refActionData.aParams[5]);
		
		fbSetPress(bExecute:= TRUE,	pPneuChannelRef:= pPneuChannelPress,nErrorId=> M_ExeAction);
		IF fbSetPress.bError THEN
			RETURN;
		END_IF
		
		IF NOT bSetPress AND fbSetPress.bBusy THEN
			bSetPress := TRUE;
			fbList.A_AddHeadValue(hList := hList, putValue := E_Action.ACTION_SetPressure);
		ELSE
			RETURN;	
		END_IF

	E_Action.ACTION_SetVacuum:
		fbSetVacuum(bExecute:= FALSE, pPneuChannelRef:= pPneuChannelVac); //eventueller Fehler wird auch zurückgesetzt
		fbSetVacuum.bAwait := DINT_TO_BOOL(refActionData.aParams[1]);
		fbSetVacuum.nValue := DINT_TO_INT(refActionData.aParams[2]);
		fbSetVacuum.nTolerancePlus := DINT_TO_INT(refActionData.aParams[3]);
		fbSetVacuum.nToleranceMinus := DINT_TO_INT(refActionData.aParams[4]);
		fbSetVacuum.tTimeout := DINT_TO_TIME(refActionData.aParams[5]);
		
		fbSetVacuum(bExecute:= TRUE, pPneuChannelRef:= pPneuChannelVac,nErrorId=> M_ExeAction);
		IF fbSetVacuum.bError THEN
			RETURN;
		END_IF
		
		IF NOT bSetVacuum AND fbSetVacuum.bBusy THEN
			bSetVacuum := TRUE;
			fbList.A_AddHeadValue(hList := hList, putValue := E_Action.ACTION_SetVacuum);
		ELSE
			RETURN;	
		END_IF

	E_Action.ACTION_SwitchPressure:
		ePressCtrl := DINT_TO_USINT(refActionData.aParams[1]);
		tPressTime := DINT_TO_TIME(refActionData.aParams[2]);
		IF ePressCtrl = E_PressCtrl.PRESSCTRL_Off OR ePressCtrl = E_PressCtrl.PRESSCTRL_PressOn 
													OR ePressCtrl = E_PressCtrl.PRESSCTRL_VacOn THEN
			IF NOT bSwitchPress THEN
				fbList.A_AddHeadValue(hList := hList, putValue := E_Action.ACTION_SwitchPressure);
				bSwitchPress := TRUE;
			END_IF
		END_IF
				
	E_Action.ACTION_PulsePressure:
		bPulseOn := DINT_TO_BOOL(refActionData.aParams[6]);
		IF bPulseOn THEN	//On
			eSwitchCtrlPhase1 := DINT_TO_USINT(refActionData.aParams[1]);
			eSwitchCtrlPhase2 := DINT_TO_USINT(refActionData.aParams[2]);
	
			IF NOT(refActionData.aParams[4] >= 1 AND refActionData.aParams[4] <= 100) THEN
				M_ExeAction := E_ErrorIdCmd.ERRORID_InvalidDutyCycle;  //Error
				RETURN;
			END_IF
			nTimePhase1 := DINT_TO_UINT(refActionData.aParams[3] / 100 * refActionData.aParams[4]); 
			nTimePhase2 := DINT_TO_UINT(refActionData.aParams[3] - nTimePhase1);
			IF NOT bPulsePress THEN
				bPulsePress := TRUE;
				fbList.A_AddHeadValue(hList := hList, putValue := E_Action.ACTION_PulsePressure);
			ELSE
				RETURN;
			END_IF
			nCurrentPulses := 0;
			nSetpointPulses := DINT_TO_UINT(refActionData.aParams[5]);
		ELSE
			RETURN;
		END_IF				

	E_Action.ACTION_PickPutPowder:
		IF NOT bPickPut THEN
			ePickPutMode := DINT_TO_USINT(refActionData.aParams[1]);
			nIntakeVac := DINT_TO_INT(refActionData.aParams[2]);
			tIntakeTime := DINT_TO_TIME(refActionData.aParams[3]);
			nHoldVac := DINT_TO_INT(refActionData.aParams[4]);
			nBlowOutPress := DINT_TO_INT(refActionData.aParams[5]);
			nBlowOutPulseTime := DINT_TO_UINT(refActionData.aParams[6]);
			nBlowOutPulses := DINT_TO_UINT(refActionData.aParams[7]);
			IF nBlowOutPulseTime = 0 OR nBlowOutPulses = 0 THEN
				RETURN;
			END_IF
			bPickPut := TRUE;
			fbList.A_AddHeadValue(hList := hList, putValue := E_Action.ACTION_PickPutPowder);
		ELSE
			RETURN;	
		END_IF
	ELSE
		M_ExeAction := SUPER^.M_ExeAction(refActionData);
		RETURN;
END_CASE

bBusy := TRUE;
eCurrentState := E_MachineState.MACHINESTATE_Active;
END_METHOD

METHOD M_GetAllProps : ERRORID
VAR_INPUT
	refCmdData : REFERENCE TO  ST_CmdData;
END_VAR
//Basisproperties lesen
SUPER^.M_GetAllProps(refCmdData);
//Specialproperties lesen
nCurrentPropIndex := nCurrentPropIndex + 1; 
IF pPneuChannelPress > 0 THEN
	refCmdData.n32Data[nCurrentPropIndex] := pPneuChannelPress^.nChannel;
ELSE
	refCmdData.n32Data[nCurrentPropIndex] := 0;
END_IF

nCurrentPropIndex := nCurrentPropIndex + 1;
IF pPneuChannelVac > 0 THEN
	refCmdData.n32Data[nCurrentPropIndex] := pPneuChannelVac^.nChannel;
ELSE
	refCmdData.n32Data[nCurrentPropIndex] := 0;
END_IF

nCurrentPropIndex := nCurrentPropIndex + 1;
refCmdData.n32Data[nCurrentPropIndex] := nDOutChanValvePress; //Digitaler Ausgangskanal MzHead Druckventil
nCurrentPropIndex := nCurrentPropIndex + 1;
refCmdData.n32Data[nCurrentPropIndex] := nDOutChanValveVac;	//Digitaler Ausgangskanal MzHead Vakuumventil
END_METHOD

METHOD M_SetAllProps : ERRORID
VAR_INPUT
	refCmdData : REFERENCE TO  ST_CmdData;
END_VAR

VAR
	nPneuChannel : USINT;
END_VAR
M_SetAllProps := SUPER^.M_SetAllProps(refCmdData);

IF M_SetAllProps > 0 THEN
	RETURN;
END_IF

//PneuChannel Druck
nCurrentPropIndex := nCurrentPropIndex + 1;
nSpecPropIndex := nCurrentPropIndex;
nPneuChannel := DINT_TO_USINT(refCmdData.n32Data[nCurrentPropIndex]);
IF NOT (nPneuChannel > 0 AND nPneuChannel <= cNoOfPneuChannels) THEN
	M_SetAllProps := E_ErrorIdObjMgmt.ERRORID_InvalidPneuChannel;
	RETURN;	
END_IF
pPneuChannelPress := ADR(aFbPneuChannel[nPneuChannel]);

//PneuChannel Vakuum
nCurrentPropIndex := nCurrentPropIndex + 1;
nPneuChannel := DINT_TO_USINT(refCmdData.n32Data[nCurrentPropIndex]);		
IF NOT (nPneuChannel > 0 AND nPneuChannel <= cNoOfPneuChannels) THEN
	M_SetAllProps := E_ErrorIdObjMgmt.ERRORID_InvalidPneuChannel;
	RETURN;	
END_IF
pPneuChannelVac := ADR(aFbPneuChannel[nPneuChannel]);

nCurrentPropIndex := nCurrentPropIndex + 1;
nDOutChanValvePress := DINT_TO_USINT(refCmdData.n32Data[nCurrentPropIndex]); //Digitaler Ausgangskanal MzHead Druckventil Pressure
IF NOT(nDOutChanValvePress >= 0 AND nDOutChanValvePress <= 7) THEN
	M_SetAllProps := E_ErrorIdObjMgmt.ERRORID_InvalidMzDOutChannel;
	RETURN;
END_IF

nCurrentPropIndex := nCurrentPropIndex + 1;
nDOutChanValveVac := DINT_TO_USINT(refCmdData.n32Data[nCurrentPropIndex]);	//Digitaler Ausgangskanal MzHead Druckventil Vacuum
IF NOT(nDOutChanValveVac >= 0 AND nDOutChanValveVac <= 7) THEN	//kann 0 sein
	M_SetAllProps := E_ErrorIdObjMgmt.ERRORID_InvalidMzDOutChannel;
	RETURN;
END_IF

pZAxisRef^.eFixedToolType := E_MzToolType.TOOL_TYPE_PowderPip;

nNoOfProps := nCurrentPropIndex + 1;
END_METHOD

METHOD M_SetSingleProp : ERRORID
VAR_INPUT
	refCmdData : REFERENCE TO  ST_CmdData;
END_VAR

VAR
	nPneuChannel : USINT;
END_VAR
IF nSpecPropIndex = refCmdData.aHeader[1] THEN	//PneuChannel Druck
	nPneuChannel := DINT_TO_USINT(refCmdData.n32Data[0]);
	IF NOT (nPneuChannel > 0 AND nPneuChannel <= cNoOfPneuChannels) THEN
		M_SetSingleProp := E_ErrorIdObjMgmt.ERRORID_InvalidPneuChannel;
		RETURN;	
	END_IF
	pPneuChannelPress := ADR(aFbPneuChannel[nPneuChannel]);
ELSIF (nSpecPropIndex + 1) = refCmdData.aHeader[1] THEN //PneuChannel Vakuum
	nPneuChannel := DINT_TO_USINT(refCmdData.n32Data[0]);
	IF NOT (nPneuChannel >= 0 AND nPneuChannel <= cNoOfPneuChannels) THEN
		M_SetSingleProp := E_ErrorIdObjMgmt.ERRORID_InvalidPneuChannel;
		RETURN;	
	END_IF
	pPneuChannelVac := ADR(aFbPneuChannel[nPneuChannel]);		
ELSIF (nSpecPropIndex + 2) = refCmdData.aHeader[1] THEN //Digitaler Ausgangskanal MzHead Druckventil
	IF refCmdData.n32Data[0] < 1 OR refCmdData.n32Data[0] > 7 THEN	//Ausgang 1-7
		M_SetSingleProp := E_ErrorIdObjMgmt.ERRORID_InvalidMzDOutChannel;
		RETURN;
	END_IF
	nDOutChanValvePress := DINT_TO_USINT(refCmdData.n32Data[0]);	
ELSIF (nSpecPropIndex + 3) = refCmdData.aHeader[1] THEN //Digitaler Ausgangskanal MzHead Vakuumventil
	IF refCmdData.n32Data[0] < 1 OR refCmdData.n32Data[0] > 7 THEN	//Ausgang 1-7
		M_SetSingleProp := E_ErrorIdObjMgmt.ERRORID_InvalidMzDOutChannel;
		RETURN;
	END_IF
	nDOutChanValveVac := DINT_TO_USINT(refCmdData.n32Data[0]);	
ELSE
	M_SetSingleProp := SUPER^.M_SetSingleProp(refCmdData);
END_IF
END_METHOD

PROPERTY P_bIsInit : BOOL
GET
P_bIsInit := bInitToolOk AND SUPER^.P_bIsInit;
END_GET
END_PROPERTY

PROPERTY P_rToolRadius : REAL
GET
VAR
	stDim : ST_3DDimension;
END_VAR
P_rToolRadius := 4000.0;
END_GET
END_PROPERTY

END_FUNCTION_BLOCK

// ---- Objects/Tools/FB_CartDispStirrer.TcPOU
FUNCTION_BLOCK FB_CartDispStirrer EXTENDS FB_CartDispenser

VAR_OUTPUT
END_VAR
VAR
	
	//Specproperties
	nPWM_Channel	: USINT;
	nStartSpeed		: UINT;
	tStartTime		: TIME;
	//****************************************Aktionsvariablen****************************************************
	
	nStateA_Stirr	: USINT;
	bStirrerOn		: BOOL;
	nStirrSpeed		: UINT;
	tStirrTimeOn	: TIME;
	tStirrTimeOff	: TIME;
	timerStirr		: TON;
	
END_VAR

A_Stirr();
SUPER^();
stProcessData.n32Data[10] := BOOL_TO_DINT(nStateA_Stirr > 0);
aObjProcData[nNotifyId] := stProcessData;

ACTION A_Stirr:
IF nPWM_Channel = 0 THEN
	RETURN;
END_IF

IF NOT bStirrerOn THEN
	timerStirr(IN:= FALSE);
	fbMultiZPWM.M_Off(nPWM_Channel);
	nStateA_Stirr := 0;
END_IF

CASE nStateA_Stirr OF
	0:	//Off
		IF bStirrerOn THEN
			nStateA_Stirr := 1;
		END_IF
		
	1:	//StartUp
		timerStirr(IN:= TRUE, PT:= tStartTime);
		IF timerStirr.Q THEN
			timerStirr(IN:= FALSE);
			IF tStirrTimeOn = T#0MS OR tStirrTimeOff = T#0MS THEN
				nStateA_Stirr := 2;
			ELSE
				nStateA_Stirr := 2;
			END_IF
		END_IF
		fbMultiZPWM.M_On(nPWM_Channel, nStartSpeed);

	2:	//ContiOn
		IF tStirrTimeOn = T#0MS OR tStirrTimeOff = T#0MS THEN
			fbMultiZPWM.M_On(nPWM_Channel, nStirrSpeed);
		ELSE
			nStateA_Stirr := 3;
		END_IF
	
	3:	//Alternating On
		IF tStirrTimeOn = T#0MS OR tStirrTimeOff = T#0MS THEN
			timerStirr(IN:= FALSE);
			nStateA_Stirr := 2;
		ELSE
			timerStirr(IN:= TRUE, PT:= tStirrTimeOn);
			IF timerStirr.Q THEN
				timerStirr(IN:= FALSE);
				fbMultiZPWM.M_Off(nPWM_Channel);
				nStateA_Stirr := 4;
			ELSE
				fbMultiZPWM.M_On(nPWM_Channel, nStirrSpeed);
			END_IF
		END_IF
	
	4:	//Alternating Off
		IF tStirrTimeOn = T#0MS OR tStirrTimeOff = T#0MS THEN
			timerStirr(IN:= FALSE);
			nStateA_Stirr := 1;
		ELSE
			timerStirr(IN:= TRUE, PT:= tStirrTimeOff);
			IF timerStirr.Q THEN
				timerStirr(IN:= FALSE);
				nStateA_Stirr := 1;
			END_IF
		END_IF
END_CASE
END_ACTION

METHOD FB_init : BOOL
VAR_INPUT
	bInitRetains : BOOL; // if TRUE, the retain variables are initialized (warm start / cold start)
	bInCopyCode : BOOL;  // if TRUE, the instance afterwards gets moved into the copy code (online change)
END_VAR
eObjectType := E_ObjectType.OBJECTTYPE_CartDispStirrer;
END_METHOD

METHOD M_CheckAction : ERRORID
VAR_INPUT
	refActionData : REFERENCE TO ST_ActionData;
	pCorrelObject	: POINTER TO FB_Object;
END_VAR
CASE refActionData.eAction OF
	(*E_Action.ACTION_CleanTip,
	E_Action.ACTION_MeasureTool,
	E_Action.ACTION_SwitchPressure, //BasicAction für ActionOnArray
	E_Action.ACTION_TeachTarget:
		RETURN;*)
ELSE
	M_CheckAction := SUPER^.M_CheckAction(refActionData, pCorrelObject);
END_CASE
END_METHOD

METHOD M_ClearAllProps
VAR_INPUT
	bIgnoreParent : BOOL; //Es wird das gesamte OD gelöscht. -> Zeiger auf Parent nicht mehr gültig!
END_VAR
nPWM_Channel := 0;
bStirrerOn := FALSE;
SUPER^.M_ClearAllProps(bIgnoreParent);
END_METHOD

METHOD M_ExeAction : ERRORID
VAR_INPUT
	refActionData : REFERENCE TO ST_ActionData;	
END_VAR
IF NOT (eCurrentState = E_MachineState.MACHINESTATE_Idle OR
	eCurrentState = E_MachineState.MACHINESTATE_Active OR
	eCurrentState = E_MachineState.MACHINESTATE_Ready) THEN
	M_ExeAction := E_ErrorIdCmd.ERRORID_InvalidState;
	RETURN;
END_IF

CASE refActionData.eAction OF
	E_Action.ACTION_StirrCartridge:
		bStirrerOn := DINT_TO_BOOL(refActionData.aParams[1]);
		nStirrSpeed := DINT_TO_UINT(refActionData.aParams[2]);
		tStirrTimeOn := DINT_TO_TIME(refActionData.aParams[3]);
		tStirrTimeOff := DINT_TO_TIME(refActionData.aParams[4]);
	ELSE
		M_ExeAction := SUPER^.M_ExeAction(refActionData);
		RETURN;
END_CASE

bBusy := TRUE;
eCurrentState := E_MachineState.MACHINESTATE_Active;
END_METHOD

METHOD M_GetAllProps : ERRORID
VAR_INPUT
	refCmdData : REFERENCE TO  ST_CmdData;
END_VAR
//Basisproperties lesen
SUPER^.M_GetAllProps(refCmdData);
//Specialproperties lesen
nCurrentPropIndex := nCurrentPropIndex + 1;
refCmdData.n32Data[nCurrentPropIndex] := nPWM_Channel;
nCurrentPropIndex := nCurrentPropIndex + 1;
refCmdData.n32Data[nCurrentPropIndex] := nStartSpeed;
nCurrentPropIndex := nCurrentPropIndex + 1;
refCmdData.n32Data[nCurrentPropIndex] := TIME_TO_DINT(tStartTime);
END_METHOD

METHOD M_SetAllProps : ERRORID
VAR_INPUT
	refCmdData : REFERENCE TO  ST_CmdData;
END_VAR

VAR
	nPneuChannel : USINT;
END_VAR
M_SetAllProps := SUPER^.M_SetAllProps(refCmdData);

IF M_SetAllProps > 0 THEN
	RETURN;
END_IF

nCurrentPropIndex := nCurrentPropIndex + 1;
nPWM_Channel := DINT_TO_USINT(refCmdData.n32Data[nCurrentPropIndex]);
IF NOT (nPWM_Channel >= 1 AND nPWM_Channel <= 2) THEN
	M_SetAllProps := E_ErrorIdObjMgmt.ERRORID_InvalidPWMChannel;
	RETURN;
END_IF
nCurrentPropIndex := nCurrentPropIndex + 1;
nStartSpeed := DINT_TO_UINT(refCmdData.n32Data[nCurrentPropIndex]);
IF NOT (nStartSpeed >= 1 AND nStartSpeed <= 1000) THEN
	M_SetAllProps := E_ErrorIdObjMgmt.ERRORID_InvalidStartSpeed;
	RETURN;
END_IF
nCurrentPropIndex := nCurrentPropIndex + 1;
tStartTime := DINT_TO_TIME(refCmdData.n32Data[nCurrentPropIndex]);

nNoOfProps := nCurrentPropIndex + 1;
END_METHOD

METHOD M_SetSingleProp : ERRORID
VAR_INPUT
	refCmdData : REFERENCE TO  ST_CmdData;
END_VAR

VAR
	nPneuChannel : USINT;
END_VAR
IF nSpecPropIndex + 4 = refCmdData.aHeader[1] THEN	//PWM-Channel
	IF (refCmdData.n32Data[0] >= 1 AND refCmdData.n32Data[0] <= 2) THEN
		nPWM_Channel := DINT_TO_USINT(refCmdData.n32Data[0]);
	ELSE
		M_SetSingleProp := E_ErrorIdObjMgmt.ERRORID_InvalidPWMChannel;
		RETURN;		
	END_IF
ELSIF nSpecPropIndex + 5 = refCmdData.aHeader[1] THEN	//StartSpeed
	IF (refCmdData.n32Data[0] >= 1 AND refCmdData.n32Data[0] <= 1000) THEN
		nStartSpeed := DINT_TO_UINT(refCmdData.n32Data[0]);
	ELSE
		M_SetSingleProp := E_ErrorIdObjMgmt.ERRORID_InvalidStartSpeed;
		RETURN;		
	END_IF
ELSIF nSpecPropIndex + 6 = refCmdData.aHeader[1] THEN	//StartTime
	tStartTime := DINT_TO_TIME(refCmdData.n32Data[0]);
ELSE
	M_SetSingleProp := SUPER^.M_SetSingleProp(refCmdData);
END_IF
END_METHOD

END_FUNCTION_BLOCK

// ---- Objects/Tools/FB_CartHolder.TcPOU
FUNCTION_BLOCK FB_CartHolder EXTENDS FB_MzTool
VAR_OUTPUT
END_VAR
VAR
	
	//Specproperties
	pFbHeaterRef		: POINTER TO FB_MZHeaterRef;

	//****************************************Aktionsvariablen****************************************************

	//Action: "HeatingCooling"
	bHeating			: BOOL;
	bCooling			: BOOL;
	nStateA_HeatingCooling	: USINT;	
	nTempSetpoint		: UINT;			//Solltemperatur Heizzone1
	nTempSetpoint2		: UINT;			//Solltemperatur Heizzone2
	bHeatingCoolingOn	: BOOL;			//Heizung bzw. Kühlung "EIN"
	nCurrentTemp		: UINT;			//Isttemperatur Heizzone1
	nCurrentTemp2		: UINT;			//Isttemperatur Heizzone2
	fbHeaterCtrl		: FB_MzHeaterControl;

END_VAR

VAR CONSTANT
	cHotTemp			: UINT := 500;	//(50°C) ab dieser Isttemperatur wird Tool als heiß betrachtet (Interlock)
	cMinHeatingTemp		: UINT := 30;	//(3°C) gilt nur für Kühlkartusche
	cMaxHeatingTemp		: UINT := 900;	//(90,0°C) gilt nur für Kühlkartusche
END_VAR

IF eCurrentState = E_MachineState.MACHINESTATE_Active THEN
	IF bHeating THEN
		A_HeatingCooling();
		IF nStateA_HeatingCooling >= 80 THEN
			IF nStateA_HeatingCooling >= 99 THEN
				bError := TRUE;
			END_IF
			bHeating := FALSE;
			nStateA_HeatingCooling := 0;
			M_RemoveListEntry(nSearchValue:= E_Action.ACTION_Heating);
		END_IF
	END_IF
	
	IF bCooling THEN
		A_HeatingCooling();
		IF nStateA_HeatingCooling >= 80 THEN
			IF nStateA_HeatingCooling >= 99 THEN
				bError := TRUE;
			END_IF
			bCooling := FALSE;
			nStateA_HeatingCooling := 0;
			M_RemoveListEntry(nSearchValue:= E_Action.ACTION_Cooling);
		END_IF
	END_IF	
END_IF

SUPER^();	//FB_MzTool aufrufen

//Prozessdaten aktualisieren
IF pFbHeaterRef > 0 THEN
	stProcessData.n32Data[7] := BOOL_TO_DINT(pFbHeaterRef^.bHeaterIsOn);
	nCurrentTemp := pFbHeaterRef^.nTemp1Actual;
	nCurrentTemp2 := pFbHeaterRef^.nTemp2Actual;
	stProcessData.n32Data[8] := nCurrentTemp;
	stProcessData.n32Data[9] := nCurrentTemp2;
END_IF

aObjProcData[nNotifyId] := stProcessData;

ACTION A_HeatingCooling:
IF nStateA_HeatingCooling = 0 THEN
	IF bHeatingCoolingOn THEN
		nStateA_HeatingCooling := 2;			
	ELSE
		nStateA_HeatingCooling := 1;
	END_IF
END_IF

//Heater ausschalten
IF nStateA_HeatingCooling = 1 THEN
	fbHeaterCtrl(bExecute:= TRUE, bHeatingOn:= FALSE, pFbHeaterRef:= pFbHeaterRef);
	IF NOT fbHeaterCtrl.bBusy THEN
		IF fbHeaterCtrl.bError THEN
			stError.ErrorId := fbHeaterCtrl.nErrorId; 
			stError.POUState := nStateA_HeatingCooling;
			nStateA_HeatingCooling := 99;
		ELSE
			nStateA_HeatingCooling := 80;	
		END_IF
		fbHeaterCtrl(bExecute:= FALSE, pFbHeaterRef:= pFbHeaterRef);
	END_IF	
END_IF

//Heater einschalten
IF nStateA_HeatingCooling = 2 THEN
	fbHeaterCtrl(bExecute:= TRUE, nTempZone1:= nTempSetpoint, nTempZone2 := nTempSetpoint2, bHeatingOn:= TRUE, pFbHeaterRef:= pFbHeaterRef);
	IF NOT fbHeaterCtrl.bBusy THEN
		IF fbHeaterCtrl.bError THEN
			stError.ErrorId := fbHeaterCtrl.nErrorId; 
			stError.POUState := nStateA_HeatingCooling;
			nStateA_HeatingCooling := 99;
		ELSE
			nStateA_HeatingCooling := 80;	
		END_IF
		fbHeaterCtrl(bExecute:= FALSE, pFbHeaterRef:= pFbHeaterRef);
	END_IF
END_IF

IF nStateA_HeatingCooling = 70 THEN
	fbHeaterCtrl(bExecute:= FALSE, pFbHeaterRef:= pFbHeaterRef);
	nStateA_HeatingCooling := 80;
END_IF


//Errorhandling
IF nStateA_HeatingCooling = 99 THEN
	stError.POU := E_POU.POU_FB_CartDispenser;
	stError.Cmd := E_Action.ACTION_Heating;
	stError.POUAction := E_POUACT.POUACT_A_Heating;	fbErrorList.M_Add(stError);
END_IF
END_ACTION

ACTION A_Reset:
//Ist noch eine Aktion aktiv?
IF nStateA_ResetSpec = 0 THEN 
	IF bHeating OR bCooling THEN
		bHeating := FALSE;
		bCooling := FALSE;
		nStateA_HeatingCooling := 0;
	END_IF
	nStateA_ResetSpec := 80;		
END_IF

SUPER^.A_Reset();
END_ACTION

ACTION A_Stop:
IF nStateA_Stop = 0 THEN
	IF (bHeating OR bCooling) AND nStateA_HeatingCooling < 70 THEN
		nStateA_HeatingCooling := 70;
	END_IF
	nStateA_Stop := 1;
END_IF

SUPER^.A_Stop();
END_ACTION

METHOD FB_init : BOOL
VAR_INPUT
	bInitRetains : BOOL; // if TRUE, the retain variables are initialized (warm start / cold start)
	bInCopyCode : BOOL;  // if TRUE, the instance afterwards gets moved into the copy code (online change)
END_VAR
eObjectType := E_ObjectType.OBJECTTYPE_CartHolder;
eObjectGroup := E_ObjectGroup.OBJECTGROUP_MzTool OR E_ObjectGroup.OBJECTGROUP_Device;
END_METHOD

METHOD M_AddChild : ERRORID
VAR_INPUT
	pObject : POINTER TO FB_Object;
	nSlotNr	: UINT;
	nIndex : INT;
END_VAR
//Der Cartridge-Holder kann folgende Objekt-Typen aufnehmen
//CartrigeDispenser, Camera, Exposure
IF pObject > 0 THEN
	IF pObject^.P_eObjectType = E_ObjectType.OBJECTTYPE_Camera OR
		pObject^.P_eObjectType = E_ObjectType.OBJECTTYPE_Exposure OR
		pObject^.P_eObjectType = E_ObjectType.OBJECTTYPE_DummyTool OR
		pObject^.P_eObjectType = E_ObjectType.OBJECTTYPE_CartDispenser OR
		pObject^.P_eObjectType = E_ObjectType.OBJECTTYPE_CartDispStirrer THEN
		M_AddChild := SUPER^.M_AddChild(pObject,nSlotNr,nIndex);
	ELSE
		M_AddChild := E_ErrorIdObjMgmt.ERRORID_InvalidParentObject;
	END_IF
ELSE
	M_AddChild := E_ErrorIdObjMgmt.ERRORID_InvalidParentObject;
END_IF
END_METHOD

METHOD M_CancelAction
VAR_INPUT
	eAction : E_Action;
END_VAR
IF eAction = E_Action.ACTION_Heating THEN
	IF (bHeating or bCooling) AND nStateA_HeatingCooling < 70 THEN
		nStateA_HeatingCooling := 70;
	END_IF
ELSE
	SUPER^.M_CancelAction(eAction);
END_IF
END_METHOD

METHOD M_CheckProcDataType : BOOL
VAR_INPUT
	eProcDataType : E_ProcDataType;
END_VAR
M_CheckProcDataType := (eProcDataType = E_ProcDataType.PROCDATATYPE_Temp1) OR (eProcDataType = E_ProcDataType.PROCDATATYPE_Temp2);
END_METHOD

METHOD M_ExeAction : ERRORID
VAR_INPUT
	refActionData : REFERENCE TO ST_ActionData;	
END_VAR
IF NOT (eCurrentState = E_MachineState.MACHINESTATE_Idle OR
	eCurrentState = E_MachineState.MACHINESTATE_Active OR
	eCurrentState = E_MachineState.MACHINESTATE_Ready) THEN
	M_ExeAction := E_ErrorIdCmd.ERRORID_InvalidState;
	RETURN;
END_IF

CASE refActionData.eAction OF
	E_Action.ACTION_Heating:
		IF NOT (bHeating OR bCooling) THEN
			nTempSetpoint := DINT_TO_UINT(refActionData.aParams[1]);
			bHeatingCoolingOn := DINT_TO_BOOL(refActionData.aParams[2]);
			IF pZAxisRef^.eFixedToolType = E_MzToolType.TOOL_TYPE_CoolingCartridge THEN
				IF nTempSetpoint >= cMinHeatingTemp AND nTempSetpoint <= cMaxHeatingTemp THEN
					bHeating := TRUE;
					fbList.A_AddHeadValue(hList := hList, putValue := E_Action.ACTION_Heating);
				ELSE
					M_ExeAction := E_ErrorIdCmd.ERRORID_InvalidHeatingTemp;
					RETURN;
				END_IF
			ELSE	//betrifft MB-Kartusche und HT-Kartusche
					//hier wird die untere Grenze der Temperaturen nicht berücksichtigt
				IF nTempSetpoint > 2500 THEN
					M_ExeAction := E_ErrorIdCmd.ERRORID_InvalidHeatingTemp;
					RETURN;
				END_IF
				nTempSetpoint2 := DINT_TO_UINT(refActionData.aParams[3]);
				IF nTempSetpoint2 > 2500 THEN
					M_ExeAction := E_ErrorIdCmd.ERRORID_InvalidHeatingTemp;
					RETURN;
				END_IF
				bHeating := TRUE;
				fbList.A_AddHeadValue(hList := hList, putValue := E_Action.ACTION_Heating);
			END_IF
		END_IF
		
	//Gab es nur in V2.0.17.x mit erster Version der Kühlkartusche
	(*E_Action.ACTION_Cooling:
		//diese Action ist nur erlaubt, wenn MzToolType "CoolingCartridge" ist
		IF pZAxisRef^.eFixedToolType = E_MzToolType.TOOL_TYPE_CoolingCartridge THEN
			IF NOT (bHeating OR bCooling) THEN
				nTempSetpoint := DINT_TO_UINT(refActionData.aParams[1]);
				bHeatingCoolingOn := DINT_TO_BOOL(refActionData.aParams[2]);
				IF nTempSetpoint >= cMinCoolingTemp AND nTempSetpoint <= cMaxCoolingTemp THEN
					bCooling := TRUE;
					fbList.A_AddHeadValue(hList := hList, putValue := E_Action.ACTION_Cooling);
				ELSE
					M_ExeAction := E_ErrorIdCmd.ERRORID_InvalidHeatingTemp;
					RETURN;	
				END_IF
			END_IF
 		ELSE
			M_ExeAction := E_ErrorIdCmd.ERRORID_InvalidAction;
			RETURN;
		END_IF*)
	ELSE
		M_ExeAction := SUPER^.M_ExeAction(refActionData);
		RETURN;
END_CASE

bBusy := TRUE;
eCurrentState := E_MachineState.MACHINESTATE_Active;
END_METHOD

METHOD M_GetAllProps : ERRORID
VAR_INPUT
	refCmdData : REFERENCE TO  ST_CmdData;
END_VAR
//Basisproperties lesen
SUPER^.M_GetAllProps(refCmdData);
//Specialproperties lesen
nCurrentPropIndex := nCurrentPropIndex + 1;
IF pZAxisRef^.eFixedToolType = E_MzToolType.TOOL_TYPE_None THEN
	refCmdData.n32Data[nCurrentPropIndex] := 0;
ELSIF pZAxisRef^.eFixedToolType = E_MzToolType.TOOL_TYPE_Cartridge THEN
	refCmdData.n32Data[nCurrentPropIndex] := E_MzHeaterType.SingleHeater;
ELSIF pZAxisRef^.eFixedToolType = E_MzToolType.TOOL_TYPE_CoolingCartridge THEN
	refCmdData.n32Data[nCurrentPropIndex] := E_MzHeaterType.HeaterCooler;	
ELSIF pZAxisRef^.eFixedToolType = E_MzToolType.TOOL_TYPE_HTCartrigde THEN
	refCmdData.n32Data[nCurrentPropIndex] := E_MzHeaterType.TwinHeater;
END_IF
END_METHOD

METHOD M_GetProcData : DINT
VAR_INPUT
	eProcDataType : E_ProcDataType;
END_VAR
IF eProcDataType = E_ProcDataType.PROCDATATYPE_Temp1 THEN
	M_GetProcData := nCurrentTemp;
ELSIF eProcDataType = E_ProcDataType.PROCDATATYPE_Temp2 THEN
	M_GetProcData := nCurrentTemp2;
ELSIF eProcDataType = E_ProcDataType.PROCDATATYPE_Press1 THEN
	M_GetProcData := stProcessData.n32Data[10];
END_IF
END_METHOD

METHOD M_SetAllProps : ERRORID
VAR_INPUT
	refCmdData : REFERENCE TO  ST_CmdData;
END_VAR
M_SetAllProps := SUPER^.M_SetAllProps(refCmdData);

IF M_SetAllProps > 0 THEN
	RETURN;
END_IF

nCurrentPropIndex := nCurrentPropIndex + 1;
pFbHeaterRef := ADR(pFbMultiZ^.aFbHeaterRef[pZAxisRef^.nChannel]);

IF refCmdData.n32Data[nCurrentPropIndex] = E_MzHeaterType.Nothing THEN
	pFbHeaterRef^.P_bHeaterFixed := FALSE;
	pFbHeaterRef := 0;
	pZAxisRef^.eFixedToolType := E_MzToolType.TOOL_TYPE_None;
ELSIF refCmdData.n32Data[nCurrentPropIndex] = E_MzHeaterType.SingleHeater THEN
	pFbHeaterRef^.P_bHeaterFixed := TRUE;
	pZAxisRef^.eFixedToolType := E_MzToolType.TOOL_TYPE_Cartridge;
ELSIF refCmdData.n32Data[nCurrentPropIndex] = E_MzHeaterType.HeaterCooler THEN
	pFbHeaterRef^.P_bHeaterFixed := TRUE;
	pZAxisRef^.eFixedToolType := E_MzToolType.TOOL_TYPE_CoolingCartridge;
	//Die Version der CoolingCartridge muss mind. 101 sein. In vorheriger Version konnte die Temperatur nicht
	//durchgehend eingestellt werden.
	IF pZAxisRef^.nToolVersion < 101 THEN
		M_SetAllProps := E_ErrorIdMultiZ.ERRORID_FirmwareCartCoolerToLow;
		RETURN;
	END_IF
ELSIF refCmdData.n32Data[nCurrentPropIndex] = E_MzHeaterType.TwinHeater THEN
	pFbHeaterRef^.P_bHeaterFixed := TRUE;
	pZAxisRef^.eFixedToolType := E_MzToolType.TOOL_TYPE_HTCartrigde;
ELSE
	M_SetAllProps := E_ErrorIdObjMgmt.ERRORID_InvalidHeaterType;
END_IF
nNoOfProps := nCurrentPropIndex + 1;
END_METHOD

PROPERTY P_bIsHot : BOOL
GET
P_bIsHot := nCurrentTemp >= cHotTemp OR nCurrentTemp2 >= cHotTemp;
END_GET
END_PROPERTY

END_FUNCTION_BLOCK

// ---- Objects/Tools/FB_Camera.TcPOU
FUNCTION_BLOCK FB_Camera EXTENDS FB_GCodeTool
VAR_INPUT
END_VAR
VAR_OUTPUT
END_VAR
VAR
	//SpecProperties
	rWorkingDistance		: REAL;
	bInvertWorkingDistance 	: BOOL;
	eLightOutput 			: E_TriggerOutput;
	nLightOutputChannel		: USINT;
	
	bCameraLightOn			: BOOL;
	
	bTakePicture			: BOOL;
	nStateA_TakePicture		: USINT;
	tDelayTakePicture		: TIME;
	timerTakePicture		: TON;
	nRequestArg1			: DINT;
	nRequestArg2			: DINT;
	nRequestArg3			: DINT;
	nRequestArg4			: DINT;	
END_VAR

IF bCameraLightOn THEN
	IF eLightOutput = E_TriggerOutput.MultiZOutput THEN
		fbMultiZDigiOut.M_On(nLightOutputChannel);
	ELSIF eLightOutput = E_TriggerOutput.MultiZPWM THEN
		fbMultiZPWM.M_On(nLightOutputChannel, 1000);
	END_IF
END_IF

IF eCurrentState = E_MachineState.MACHINESTATE_Active THEN
	IF bTakePicture THEN
		A_TakePicture();
		IF nStateA_TakePicture = 80 THEN
			nStateA_TakePicture := 0;
			bTakePicture := FALSE;
			M_RemoveListEntry(nSearchValue:= E_Action.ACTION_TakePicture);
		END_IF
	END_IF	
END_IF

SUPER^();

stProcessData.n32Data[7] := BOOL_TO_DINT(bCameraLightOn);
aObjProcData[nNotifyId] := stProcessData;

ACTION A_Reset:
nStateA_ResetSpec := 80;
SUPER^.A_Reset();
END_ACTION

ACTION A_Stop:
IF nStateA_Stop = 0 THEN
	IF bTakePicture AND nStateA_TakePicture < 70 THEN
		nStateA_TakePicture := 70;
	END_IF
	nStateA_Stop := 1;
END_IF

SUPER^.A_Stop();
END_ACTION

ACTION A_TakePicture:
IF nStateA_TakePicture = 0 THEN //Timer starten
	timerTakePicture(IN:= TRUE, PT:= tDelayTakePicture);
	IF timerTakePicture.Q THEN
		timerTakePicture(IN:= FALSE);
		stInterResponse.eInteractMessageType := E_InteractMessageType.INTERACTMES_NONE;
		stInteractRequest.eInteractMessageType := E_InteractMessageType.INTERACTMES_WaitForUser;
		stInteractRequest.nObjectId := nObjectID;
		stInteractRequest.nArg1 := nRequestArg1;
		stInteractRequest.nArg2 := nRequestArg2;
		stInteractRequest.nArg3 := nRequestArg3;
		stInteractRequest.nArg4 := nRequestArg4;
		nStateA_TakePicture := 1;
	END_IF
ELSIF nStateA_TakePicture = 1 THEN //Auf InteractResponse warten
	IF stInterResponse.eInteractMessageType = E_InteractMessageType.INTERACTMES_Continue OR 
							stInterResponse.eInteractMessageType = E_InteractMessageType.INTERACTMES_Cancel THEN
		stInteractRequest.eInteractMessageType := E_InteractMessageType.INTERACTMES_NONE;
		nStateA_TakePicture := 80;
	END_IF
ELSIF nStateA_TakePicture = 70 THEN //Abbrechen
	timerTakePicture(IN:= FALSE);
	stInteractRequest.eInteractMessageType := E_InteractMessageType.INTERACTMES_NONE;
	nStateA_TakePicture := 80;
END_IF
END_ACTION

METHOD FB_init : BOOL
VAR_INPUT
	bInitRetains : BOOL; // if TRUE, the retain variables are initialized (warm start / cold start)
	bInCopyCode : BOOL;  // if TRUE, the instance afterwards gets moved into the copy code (online change)
END_VAR
eObjectType := E_ObjectType.OBJECTTYPE_Camera;
eObjectGroup := E_ObjectGroup.OBJECTGROUP_MzTool OR E_ObjectGroup.OBJECTGROUP_Device;
END_METHOD

METHOD M_AddChild : ERRORID
VAR_INPUT
	pObject : POINTER TO FB_Object;
	nSlotNr	: UINT;	
	nIndex : INT;
END_VAR
//Kann folgende Objekte aufnehmen:
//Camera, Exposure
IF pObject > 0 THEN
	IF pObject^.P_eObjectType = E_ObjectType.OBJECTTYPE_Camera OR
		pObject^.P_eObjectType = E_ObjectType.OBJECTTYPE_DummyTool OR
		pObject^.P_eObjectType = E_ObjectType.OBJECTTYPE_Exposure THEN
		M_AddChild := SUPER^.M_AddChild(pObject,nSlotNr,nIndex);
	ELSE
		M_AddChild := E_ErrorIdObjMgmt.ERRORID_InvalidParentObject;
	END_IF
ELSE
	M_AddChild := E_ErrorIdObjMgmt.ERRORID_InvalidParentObject;
END_IF
END_METHOD

METHOD M_CancelAction
VAR_INPUT
	eAction : E_Action;
END_VAR
IF eAction = E_Action.ACTION_TakePicture THEN
	IF bTakePicture AND nStateA_TakePicture < 70 THEN
		nStateA_TakePicture := 70;
	END_IF
ELSE
	SUPER^.M_CancelAction(eAction);
END_IF
END_METHOD

METHOD M_CheckAction : ERRORID
VAR_INPUT
	refActionData 	: REFERENCE TO ST_ActionData;
	pCorrelObject	: POINTER TO FB_Object;
END_VAR

VAR
	pTarget : POINTER TO FB_TargetBase;
	pRack	: POINTER TO FB_Rack;
	pSlot	: POINTER TO FB_PieceSlot;
END_VAR
IF refActionData.eAction = E_Action.ACTION_TakePicture THEN
	RETURN;
ELSE
	M_CheckAction := SUPER^.M_CheckAction(refActionData, pCorrelObject);
END_IF
END_METHOD

METHOD M_ExeAction : ERRORID
VAR_INPUT
	refActionData : REFERENCE TO ST_ActionData;	
END_VAR
IF NOT (eCurrentState = E_MachineState.MACHINESTATE_Idle OR
	eCurrentState = E_MachineState.MACHINESTATE_Active OR
	eCurrentState = E_MachineState.MACHINESTATE_Ready) THEN
	M_ExeAction := E_ErrorIdCmd.ERRORID_InvalidState;
	RETURN;
END_IF

IF refActionData.eAction = E_Action.ACTION_SwitchLight THEN
	bCameraLightOn := DINT_TO_BOOL(refActionData.aParams[1]);
ELSIF refActionData.eAction = E_Action.ACTION_TakePicture THEN
	IF NOT bTakePicture THEN
		tDelayTakePicture := DINT_TO_TIME(refActionData.aParams[1]);
		nRequestArg1 := refActionData.aParams[2];
		nRequestArg2 := refActionData.aParams[3];
		nRequestArg3 := refActionData.aParams[4];
		nRequestArg4 := refActionData.aParams[5];
		
		fbList.A_AddHeadValue(hList := hList, putValue := E_Action.ACTION_TakePicture);
		bTakePicture := TRUE;
	END_IF
ELSE
	M_ExeAction := SUPER^.M_ExeAction(refActionData);
	RETURN;	
END_IF

bBusy := TRUE;
eCurrentState := E_MachineState.MACHINESTATE_Active;
END_METHOD

